LIN {X 0,Y 465.142,Z 330.415,A -85,B 0,C 180,E1 -14982.121,E2 -14982.121} C_VEL
LIN {X 0,Y 468.433,Z 327.76,A -85,B 0,C 180,E1 -14982.417,E2 -14982.417} C_VEL
LIN {X 0,Y 473.439,Z 325.91,A -85,B 0,C 180,E1 -14983.014,E2 -14983.014} C_VEL
LIN {X 0,Y 476.656,Z 325.887,A -85,B 0,C 180,E1 -14983.476,E2 -14983.476} C_VEL
LIN {X 0,Y 482.321,Z 341.882,A -85,B 0,C 180,E1 -14985.491,E2 -14985.491} C_VEL
LIN {X 0,Y 481.738,Z 369.053,A -85,B 0,C 180,E1 -14987.374,E2 -14987.374} C_VEL
LIN {X 0,Y 476.688,Z 392.56,A -85,B 0,C 180,E1 -14988.235,E2 -14988.235} C_VEL
LIN {X 0,Y 472.973,Z 475.5,A -85,B 0,C 180,E1 -14989.59,E2 -14989.59} C_VEL
LIN {X 0,Y 468.98,Z 538.697,A -85,B 0,C 180,E1 -14990.825,E2 -14990.825} C_VEL
LIN {X 0,Y 463.668,Z 606.761,A -85,B 0,C 180,E1 -14992.375,E2 -14992.375} C_VEL
LIN {X 0,Y 460.239,Z 651.951,A -85,B 0,C 180,E1 -14993.579,E2 -14993.579} C_VEL
LIN {X 0,Y 458.656,Z 674.727,A -85,B 0,C 180,E1 -14994.346,E2 -14994.346} C_VEL
LIN {X 0,Y 456.595,Z 696.121,A -85,B 0,C 180,E1 -14995.294,E2 -14995.294} C_VEL
LIN {X 0,Y 454.077,Z 716.813,A -85,B 0,C 180,E1 -14996.447,E2 -14996.447} C_VEL
LIN {X 0,Y 452.526,Z 727.999,A -85,B 0,C 180,E1 -14997.18,E2 -14997.18} C_VEL
LIN {X 0,Y 450.699,Z 734.854,A -85,B 0,C 180,E1 -14997.592,E2 -14997.592} C_VEL
LIN {X 0,Y 442.928,Z 751.978,A -85,B 0,C 180,E1 -14998.507,E2 -14998.507} C_VEL
LIN {X 0,Y 440.936,Z 758.361,A -85,B 0,C 180,E1 -14999.008,E2 -14999.008} C_VEL
LIN {X 0,Y 437.431,Z 776.665,A -85,B 0,C 180,E1 -15000.864,E2 -15000.864} C_VEL
LIN {X 0,Y 433.922,Z 793.74,A -85,B 0,C 180,E1 -15002.928,E2 -15002.928} C_VEL
LIN {X 0,Y 430.589,Z 809.209,A -85,B 0,C 180,E1 -15005.146,E2 -15005.146} C_VEL
LIN {X 0,Y 427.587,Z 822.933,A -85,B 0,C 180,E1 -15007.472,E2 -15007.472} C_VEL
LIN {X 0,Y 424.814,Z 835.676,A -85,B 0,C 180,E1 -15010.045,E2 -15010.045} C_VEL
LIN {X 0,Y 422.444,Z 846.943,A -85,B 0,C 180,E1 -15012.79,E2 -15012.79} C_VEL
LIN {X 0,Y 420.551,Z 856.578,A -85,B 0,C 180,E1 -15015.684,E2 -15015.684} C_VEL
LIN {X 0,Y 419.196,Z 864.185,A -85,B 0,C 180,E1 -15018.581,E2 -15018.581} C_VEL
LIN {X 0,Y 418.339,Z 869.705,A -85,B 0,C 180,E1 -15021.339,E2 -15021.339} C_VEL
LIN {X 0,Y 417.806,Z 873.843,A -85,B 0,C 180,E1 -15024.231,E2 -15024.231} C_VEL
LIN {X 0,Y 417.544,Z 876.277,A -85,B 0,C 180,E1 -15026.98,E2 -15026.98} C_VEL
LIN {X 0,Y 417.459,Z 877.198,A -85,B 0,C 180,E1 -15029.863,E2 -15029.863} C_VEL
LIN {X 0,Y 417.51,Z 876.519,A -85,B 0,C 180,E1 -15032.608,E2 -15032.608} C_VEL
LIN {X 0,Y 417.764,Z 874.258,A -85,B 0,C 180,E1 -15035.494,E2 -15035.494} C_VEL
LIN {X 0,Y 418.227,Z 870.613,A -85,B 0,C 180,E1 -15038.247,E2 -15038.247} C_VEL
LIN {X 0,Y 419.071,Z 865.05,A -85,B 0,C 180,E1 -15041.143,E2 -15041.143} C_VEL
LIN {X 0,Y 420.276,Z 858.016,A -85,B 0,C 180,E1 -15043.906,E2 -15043.906} C_VEL
LIN {X 0,Y 421.971,Z 849.236,A -85,B 0,C 180,E1 -15046.661,E2 -15046.661} C_VEL
LIN {X 0,Y 424.212,Z 838.486,A -85,B 0,C 180,E1 -15049.411,E2 -15049.411} C_VEL
LIN {X 0,Y 426.882,Z 826.191,A -85,B 0,C 180,E1 -15052.01,E2 -15052.01} C_VEL
LIN {X 0,Y 429.757,Z 813.215,A -85,B 0,C 180,E1 -15054.319,E2 -15054.319} C_VEL
LIN {X 0,Y 433.075,Z 797.976,A -85,B 0,C 180,E1 -15056.61,E2 -15056.61} C_VEL
LIN {X 0,Y 436.501,Z 781.676,A -85,B 0,C 180,E1 -15058.677,E2 -15058.677} C_VEL
LIN {X 0,Y 440.028,Z 763.676,A -85,B 0,C 180,E1 -15060.597,E2 -15060.597} C_VEL
LIN {X 0,Y 443.454,Z 744.549,A -85,B 0,C 180,E1 -15062.302,E2 -15062.302} C_VEL
LIN {X 0,Y 446.63,Z 724.241,A -85,B 0,C 180,E1 -15063.802,E2 -15063.802} C_VEL
LIN {X 0,Y 449.363,Z 703.738,A -85,B 0,C 180,E1 -15065.035,E2 -15065.035} C_VEL
LIN {X 0,Y 451.591,Z 682.841,A -85,B 0,C 180,E1 -15066.044,E2 -15066.044} C_VEL
LIN {X 0,Y 453.312,Z 661.563,A -85,B 0,C 180,E1 -15066.837,E2 -15066.837} C_VEL
LIN {X 0,Y 456.433,Z 619.357,A -85,B 0,C 180,E1 -15068.038,E2 -15068.038} C_VEL
LIN {X 0,Y 462.05,Z 551.52,A -85,B 0,C 180,E1 -15069.647,E2 -15069.647} C_VEL
LIN {X 0,Y 466.509,Z 485.901,A -85,B 0,C 180,E1 -15070.975,E2 -15070.975} C_VEL
LIN {X 0,Y 469.976,Z 414.611,A -85,B 0,C 180,E1 -15072.175,E2 -15072.175} C_VEL
LIN {X 0,Y 471.052,Z 393.311,A -85,B 0,C 180,E1 -15072.537,E2 -15072.537} C_VEL
LIN {X 0,Y 476.185,Z 369.743,A -85,B 0,C 180,E1 -15073.439,E2 -15073.439} C_VEL
LIN {X 0,Y 476.556,Z 345.293,A -85,B 0,C 180,E1 -15075.172,E2 -15075.172} C_VEL
LIN {X 0,Y 469.126,Z 324.998,A -85,B 0,C 180,E1 -15077.825,E2 -15077.825} C_VEL
LIN {X 0,Y 462.685,Z 309.482,A -85,B 0,C 180,E1 -15080.071,E2 -15080.071} C_VEL
LIN {X 0,Y 456.022,Z 295.191,A -85,B 0,C 180,E1 -15082.33,E2 -15082.33} C_VEL
LIN {X 0,Y 447.821,Z 279.246,A -85,B 0,C 180,E1 -15085.138,E2 -15085.138} C_VEL
LIN {X 0,Y 439.708,Z 265.393,A -85,B 0,C 180,E1 -15087.851,E2 -15087.851} C_VEL
LIN {X 0,Y 435.741,Z 259.224,A -85,B 0,C 180,E1 -15089.222,E2 -15089.222} C_VEL
LIN {X 0,Y 433.247,Z 255.233,A -85,B 0,C 180,E1 -15090.099,E2 -15090.099} C_VEL
LIN {X 0,Y 430.503,Z 250.807,A -85,B 0,C 180,E1 -15091.112,E2 -15091.112} C_VEL
LIN {X 0,Y 427.306,Z 246.461,A -85,B 0,C 180,E1 -15092.247,E2 -15092.247} C_VEL
LIN {X 0,Y 426.374,Z 244.715,A -85,B 0,C 180,E1 -15092.636,E2 -15092.636} C_VEL
LIN {X 0,Y 423.833,Z 241.89,A -85,B 0,C 180,E1 -15093.52,E2 -15093.52} C_VEL
LIN {X 0,Y 422.541,Z 239.071,A -85,B 0,C 180,E1 -15094.113,E2 -15094.113} C_VEL
LIN {X 0,Y 419.683,Z 236.312,A -85,B 0,C 180,E1 -15095.133,E2 -15095.133} C_VEL
LIN {X 0,Y 418.562,Z 233.254,A -85,B 0,C 180,E1 -15095.739,E2 -15095.739} C_VEL
LIN {X 0,Y 418.538,Z 233.089,A -85,B 0,C 180,E1 -15099.47,E2 -15099.47} C_VEL
LIN {X 0,Y 418.533,Z 233.058,A -85,B 0,C 180,E1 -15103.34,E2 -15103.34} C_VEL
LIN {X 0,Y 418.534,Z 233.043,A -85,B 0,C 180,E1 -15107.163,E2 -15107.163} C_VEL
LIN {X 0,Y 418.54,Z 233.095,A -85,B 0,C 180,E1 -15111.067,E2 -15111.067} C_VEL
LIN {X 0,Y 418.532,Z 233.045,A -85,B 0,C 180,E1 -15114.929,E2 -15114.929} C_VEL
LIN {X 0,Y 418.529,Z 233.064,A -85,B 0,C 180,E1 -15118.768,E2 -15118.768} C_VEL
LIN {X 0,Y 418.52,Z 233.07,A -85,B 0,C 180,E1 -15122.602,E2 -15122.602} C_VEL
LIN {X 0,Y 418.513,Z 233.043,A -85,B 0,C 180,E1 -15126.447,E2 -15126.447} C_VEL
LIN {X 0,Y 418.52,Z 233.1,A -85,B 0,C 180,E1 -15130.322,E2 -15130.322} C_VEL
LIN {X 0,Y 418.52,Z 233.096,A -85,B 0,C 180,E1 -15134.246,E2 -15134.246} C_VEL
LIN {X 0,Y 418.525,Z 233.086,A -85,B 0,C 180,E1 -15138.094,E2 -15138.094} C_VEL
LIN {X 0,Y 418.533,Z 233.168,A -85,B 0,C 180,E1 -15138.928,E2 -15138.928} C_VEL
LIN {X 0,Y 419.796,Z 236.493,A -85,B 0,C 180,E1 -15139.624,E2 -15139.624} C_VEL
LIN {X 0,Y 421.099,Z 238.531,A -85,B 0,C 180,E1 -15140.139,E2 -15140.139} C_VEL
LIN {X 0,Y 423.255,Z 242.427,A -85,B 0,C 180,E1 -15141.044,E2 -15141.044} C_VEL
LIN {X 0,Y 430.88,Z 257.106,A -85,B 0,C 180,E1 -15144.252,E2 -15144.252} C_VEL
LIN {X 0,Y 439.608,Z 273.969,A -85,B 0,C 180,E1 -15147.646,E2 -15147.646} C_VEL
LIN {X 0,Y 449.782,Z 294.439,A -85,B 0,C 180,E1 -15151.345,E2 -15151.345} C_VEL
LIN {X 0,Y 459.809,Z 315.283,A -85,B 0,C 180,E1 -15154.732,E2 -15154.732} C_VEL
LIN {X 0,Y 464.788,Z 325.491,A -85,B 0,C 180,E1 -15156.233,E2 -15156.233} C_VEL
LIN {X 0,Y 480.323,Z 350.017,A -85,B 0,C 180,E1 -15158.475,E2 -15158.475} C_VEL
LIN {X 0,Y 480.604,Z 356.269,A -85,B 0,C 180,E1 -15158.658,E2 -15158.658} C_VEL
LIN {X 0,Y 466.182,Z 601.705,A -85,B 0,C 180,E1 -15163.233,E2 -15163.233} C_VEL
LIN {X 0,Y 461.361,Z 693.458,A -85,B 0,C 180,E1 -15164.963,E2 -15164.963} C_VEL
LIN {X 0,Y 459.117,Z 717.943,A -85,B 0,C 180,E1 -15165.63,E2 -15165.63} C_VEL
LIN {X 0,Y 456.209,Z 743.457,A -85,B 0,C 180,E1 -15166.552,E2 -15166.552} C_VEL
LIN {X 0,Y 453.173,Z 765.825,A -85,B 0,C 180,E1 -15167.576,E2 -15167.576} C_VEL
LIN {X 0,Y 449.498,Z 789.387,A -85,B 0,C 180,E1 -15168.904,E2 -15168.904} C_VEL
LIN {X 0,Y 445.801,Z 811.052,A -85,B 0,C 180,E1 -15170.358,E2 -15170.358} C_VEL
LIN {X 0,Y 441.915,Z 831.707,A -85,B 0,C 180,E1 -15172.017,E2 -15172.017} C_VEL
LIN {X 0,Y 437.866,Z 852.231,A -85,B 0,C 180,E1 -15173.938,E2 -15173.938} C_VEL
LIN {X 0,Y 434.211,Z 870.106,A -85,B 0,C 180,E1 -15175.894,E2 -15175.894} C_VEL
LIN {X 0,Y 430.262,Z 889.208,A -85,B 0,C 180,E1 -15178.318,E2 -15178.318} C_VEL
LIN {X 0,Y 426.966,Z 905.358,A -85,B 0,C 180,E1 -15180.696,E2 -15180.696} C_VEL
LIN {X 0,Y 423.914,Z 920.881,A -85,B 0,C 180,E1 -15183.375,E2 -15183.375} C_VEL
LIN {X 0,Y 421.465,Z 934.402,A -85,B 0,C 180,E1 -15186.066,E2 -15186.066} C_VEL
LIN {X 0,Y 419.512,Z 946.432,A -85,B 0,C 180,E1 -15188.906,E2 -15188.906} C_VEL
LIN {X 0,Y 418.139,Z 956.77,A -85,B 0,C 180,E1 -15191.744,E2 -15191.744} C_VEL
LIN {X 0,Y 417.219,Z 965.635,A -85,B 0,C 180,E1 -15194.715,E2 -15194.715} C_VEL
LIN {X 0,Y 416.734,Z 972.905,A -85,B 0,C 180,E1 -15197.67,E2 -15197.67} C_VEL
LIN {X 0,Y 416.585,Z 978.694,A -85,B 0,C 180,E1 -15200.746,E2 -15200.746} C_VEL
LIN {X 0,Y 416.629,Z 982.359,A -85,B 0,C 180,E1 -15203.385,E2 -15203.385} C_VEL
LIN {X 0,Y 416.736,Z 985.143,A -85,B 0,C 180,E1 -15206.423,E2 -15206.423} C_VEL
LIN {X 0,Y 416.795,Z 986.147,A -85,B 0,C 180,E1 -15209.313,E2 -15209.313} C_VEL
LIN {X 0,Y 416.792,Z 985.858,A -85,B 0,C 180,E1 -15211.925,E2 -15211.925} C_VEL
LIN {X 0,Y 416.657,Z 984.108,A -85,B 0,C 180,E1 -15214.956,E2 -15214.956} C_VEL
LIN {X 0,Y 416.576,Z 980.619,A -85,B 0,C 180,E1 -15218.003,E2 -15218.003} C_VEL
LIN {X 0,Y 416.588,Z 976.376,A -85,B 0,C 180,E1 -15220.65,E2 -15220.65} C_VEL
LIN {X 0,Y 416.89,Z 969.637,A -85,B 0,C 180,E1 -15223.878,E2 -15223.878} C_VEL
LIN {X 0,Y 417.582,Z 961.789,A -85,B 0,C 180,E1 -15226.842,E2 -15226.842} C_VEL
LIN {X 0,Y 418.851,Z 951.921,A -85,B 0,C 180,E1 -15229.961,E2 -15229.961} C_VEL
LIN {X 0,Y 420.695,Z 940.588,A -85,B 0,C 180,E1 -15232.941,E2 -15232.941} C_VEL
LIN {X 0,Y 423.28,Z 927.489,A -85,B 0,C 180,E1 -15235.914,E2 -15235.914} C_VEL
LIN {X 0,Y 426.486,Z 912.889,A -85,B 0,C 180,E1 -15238.736,E2 -15238.736} C_VEL
LIN {X 0,Y 430.666,Z 895.41,A -85,B 0,C 180,E1 -15241.649,E2 -15241.649} C_VEL
LIN {X 0,Y 435.032,Z 878.269,A -85,B 0,C 180,E1 -15244.112,E2 -15244.112} C_VEL
LIN {X 0,Y 439.906,Z 859.257,A -85,B 0,C 180,E1 -15246.461,E2 -15246.461} C_VEL
LIN {X 0,Y 445.064,Z 839.529,A -85,B 0,C 180,E1 -15248.572,E2 -15248.572} C_VEL
LIN {X 0,Y 450.442,Z 818.443,A -85,B 0,C 180,E1 -15250.488,E2 -15250.488} C_VEL
LIN {X 0,Y 455.993,Z 795.957,A -85,B 0,C 180,E1 -15252.228,E2 -15252.228} C_VEL
LIN {X 0,Y 461.455,Z 772.834,A -85,B 0,C 180,E1 -15253.727,E2 -15253.727} C_VEL
LIN {X 0,Y 466.711,Z 748.74,A -85,B 0,C 180,E1 -15255.009,E2 -15255.009} C_VEL
LIN {X 0,Y 471.508,Z 724.263,A -85,B 0,C 180,E1 -15256.051,E2 -15256.051} C_VEL
LIN {X 0,Y 476.08,Z 697.875,A -85,B 0,C 180,E1 -15256.912,E2 -15256.912} C_VEL
LIN {X 0,Y 481.22,Z 660.217,A -85,B 0,C 180,E1 -15257.828,E2 -15257.828} C_VEL
LIN {X 0,Y 489.533,Z 604.335,A -85,B 0,C 180,E1 -15259.157,E2 -15259.157} C_VEL
LIN {X 0,Y 500.202,Z 547.443,A -85,B 0,C 180,E1 -15260.549,E2 -15260.549} C_VEL
LIN {X 0,Y 508.93,Z 508.11,A -85,B 0,C 180,E1 -15261.532,E2 -15261.532} C_VEL
LIN {X 0,Y 504.603,Z 526.167,A -85,B 0,C 180,E1 -15262.441,E2 -15262.441} C_VEL
LIN {X 0,Y 481.706,Z 630.182,A -85,B 0,C 180,E1 -15265.508,E2 -15265.508} C_VEL
LIN {X 0,Y 469.101,Z 693.847,A -85,B 0,C 180,E1 -15267.556,E2 -15267.556} C_VEL
LIN {X 0,Y 463.766,Z 717.456,A -85,B 0,C 180,E1 -15268.55,E2 -15268.55} C_VEL
LIN {X 0,Y 458.09,Z 740.922,A -85,B 0,C 180,E1 -15269.815,E2 -15269.815} C_VEL
LIN {X 0,Y 452.388,Z 763.754,A -85,B 0,C 180,E1 -15271.339,E2 -15271.339} C_VEL
LIN {X 0,Y 447.011,Z 785.108,A -85,B 0,C 180,E1 -15273.066,E2 -15273.066} C_VEL
LIN {X 0,Y 442.238,Z 804.171,A -85,B 0,C 180,E1 -15274.917,E2 -15274.917} C_VEL
LIN {X 0,Y 437.83,Z 821.686,A -85,B 0,C 180,E1 -15276.942,E2 -15276.942} C_VEL
LIN {X 0,Y 433.913,Z 837.047,A -85,B 0,C 180,E1 -15279.073,E2 -15279.073} C_VEL
LIN {X 0,Y 430.445,Z 850.31,A -85,B 0,C 180,E1 -15281.303,E2 -15281.303} C_VEL
LIN {X 0,Y 427.606,Z 860.933,A -85,B 0,C 180,E1 -15283.481,E2 -15283.481} C_VEL
LIN {X 0,Y 425.193,Z 869.743,A -85,B 0,C 180,E1 -15285.705,E2 -15285.705} C_VEL
LIN {X 0,Y 423.039,Z 877.204,A -85,B 0,C 180,E1 -15288.133,E2 -15288.133} C_VEL
LIN {X 0,Y 421.42,Z 882.367,A -85,B 0,C 180,E1 -15290.44,E2 -15290.44} C_VEL
LIN {X 0,Y 420.191,Z 885.911,A -85,B 0,C 180,E1 -15292.755,E2 -15292.755} C_VEL
LIN {X 0,Y 419.213,Z 887.887,A -85,B 0,C 180,E1 -15295.211,E2 -15295.211} C_VEL
LIN {X 0,Y 418.581,Z 888.17,A -85,B 0,C 180,E1 -15297.536,E2 -15297.536} C_VEL
LIN {X 0,Y 418.161,Z 886.727,A -85,B 0,C 180,E1 -15300,E2 -15300} C_VEL
LIN {X 0,Y 417.948,Z 883.54,A -85,B 0,C 180,E1 -15302.468,E2 -15302.468} C_VEL
LIN {X 0,Y 417.955,Z 878.555,A -85,B 0,C 180,E1 -15304.941,E2 -15304.941} C_VEL
LIN {X 0,Y 418.197,Z 871.701,A -85,B 0,C 180,E1 -15307.418,E2 -15307.418} C_VEL
LIN {X 0,Y 418.711,Z 862.825,A -85,B 0,C 180,E1 -15309.901,E2 -15309.901} C_VEL
LIN {X 0,Y 419.516,Z 852.331,A -85,B 0,C 180,E1 -15312.255,E2 -15312.255} C_VEL
LIN {X 0,Y 420.579,Z 840.438,A -85,B 0,C 180,E1 -15314.456,E2 -15314.456} C_VEL
LIN {X 0,Y 421.988,Z 826.127,A -85,B 0,C 180,E1 -15316.661,E2 -15316.661} C_VEL
LIN {X 0,Y 423.658,Z 810.108,A -85,B 0,C 180,E1 -15318.722,E2 -15318.722} C_VEL
LIN {X 0,Y 425.556,Z 792.28,A -85,B 0,C 180,E1 -15320.637,E2 -15320.637} C_VEL
LIN {X 0,Y 427.535,Z 773.248,A -85,B 0,C 180,E1 -15322.337,E2 -15322.337} C_VEL
LIN {X 0,Y 429.463,Z 754.068,A -85,B 0,C 180,E1 -15323.753,E2 -15323.753} C_VEL
LIN {X 0,Y 431.425,Z 733.007,A -85,B 0,C 180,E1 -15325.014,E2 -15325.014} C_VEL
LIN {X 0,Y 433.222,Z 711.178,A -85,B 0,C 180,E1 -15326.047,E2 -15326.047} C_VEL
LIN {X 0,Y 434.895,Z 687.679,A -85,B 0,C 180,E1 -15326.879,E2 -15326.879} C_VEL
LIN {X 0,Y 437.042,Z 646.566,A -85,B 0,C 180,E1 -15327.878,E2 -15327.878} C_VEL
LIN {X 0,Y 444.712,Z 506.022,A -85,B 0,C 180,E1 -15331.093,E2 -15331.093} C_VEL
LIN {X 0,Y 439.779,Z 438.733,A -85,B 0,C 180,E1 -15333.306,E2 -15333.306} C_VEL
LIN {X 0,Y 445.969,Z 387.644,A -85,B 0,C 180,E1 -15337.489,E2 -15337.489} C_VEL
LIN {X 0,Y 451.691,Z 344.172,A -85,B 0,C 180,E1 -15341.064,E2 -15341.064} C_VEL
LIN {X 0,Y 453.675,Z 344.144,A -85,B 0,C 180,E1 -15341.391,E2 -15341.391} C_VEL
LIN {X 0,Y 456.593,Z 342.501,A -85,B 0,C 180,E1 -15341.738,E2 -15341.738} C_VEL
LIN {X 0,Y 459.898,Z 339.563,A -85,B 0,C 180,E1 -15342.04,E2 -15342.04} C_VEL
LIN {X 0,Y 463.43,Z 338.215,A -85,B 0,C 180,E1 -15342.48,E2 -15342.48} C_VEL
LIN {X 0,Y 468.257,Z 334.771,A -85,B 0,C 180,E1 -15342.936,E2 -15342.936} C_VEL
LIN {X 0,Y 472.208,Z 333.263,A -85,B 0,C 180,E1 -15343.4,E2 -15343.4} C_VEL
LIN {X 0,Y 476.586,Z 346.018,A -85,B 0,C 180,E1 -15345.006,E2 -15345.006} C_VEL
LIN {X 0,Y 476.081,Z 370.363,A -85,B 0,C 180,E1 -15346.707,E2 -15346.707} C_VEL
LIN {X 0,Y 470.702,Z 395.368,A -85,B 0,C 180,E1 -15347.619,E2 -15347.619} C_VEL
LIN {X 0,Y 466.885,Z 477.849,A -85,B 0,C 180,E1 -15348.979,E2 -15348.979} C_VEL
LIN {X 0,Y 462.789,Z 540.682,A -85,B 0,C 180,E1 -15350.221,E2 -15350.221} C_VEL
LIN {X 0,Y 457.359,Z 607.896,A -85,B 0,C 180,E1 -15351.773,E2 -15351.773} C_VEL
LIN {X 0,Y 453.808,Z 652.838,A -85,B 0,C 180,E1 -15352.992,E2 -15352.992} C_VEL
LIN {X 0,Y 452.145,Z 676.013,A -85,B 0,C 180,E1 -15353.781,E2 -15353.781} C_VEL
LIN {X 0,Y 450.073,Z 696.948,A -85,B 0,C 180,E1 -15354.716,E2 -15354.716} C_VEL
LIN {X 0,Y 447.372,Z 718.396,A -85,B 0,C 180,E1 -15355.927,E2 -15355.927} C_VEL
LIN {X 0,Y 444.251,Z 739.171,A -85,B 0,C 180,E1 -15357.381,E2 -15357.381} C_VEL
LIN {X 0,Y 440.936,Z 758.361,A -85,B 0,C 180,E1 -15359.008,E2 -15359.008} C_VEL
LIN {X 0,Y 438.931,Z 764.725,A -85,B 0,C 180,E1 -15359.533,E2 -15359.533} C_VEL
LIN {X 0,Y 430.735,Z 780.584,A -85,B 0,C 180,E1 -15360.754,E2 -15360.754} C_VEL
LIN {X 0,Y 428.649,Z 786.403,A -85,B 0,C 180,E1 -15361.374,E2 -15361.374} C_VEL
LIN {X 0,Y 425.203,Z 802.108,A -85,B 0,C 180,E1 -15363.462,E2 -15363.462} C_VEL
LIN {X 0,Y 421.843,Z 816.908,A -85,B 0,C 180,E1 -15365.791,E2 -15365.791} C_VEL
LIN {X 0,Y 418.786,Z 830.224,A -85,B 0,C 180,E1 -15368.28,E2 -15368.28} C_VEL
LIN {X 0,Y 415.99,Z 842.599,A -85,B 0,C 180,E1 -15371.065,E2 -15371.065} C_VEL
LIN {X 0,Y 413.787,Z 852.799,A -85,B 0,C 180,E1 -15373.866,E2 -15373.866} C_VEL
LIN {X 0,Y 412.078,Z 861.435,A -85,B 0,C 180,E1 -15376.815,E2 -15376.815} C_VEL
LIN {X 0,Y 410.917,Z 867.862,A -85,B 0,C 180,E1 -15379.626,E2 -15379.626} C_VEL
LIN {X 0,Y 410.156,Z 872.891,A -85,B 0,C 180,E1 -15382.576,E2 -15382.576} C_VEL
LIN {X 0,Y 409.729,Z 876.243,A -85,B 0,C 180,E1 -15385.521,E2 -15385.521} C_VEL
LIN {X 0,Y 409.54,Z 877.981,A -85,B 0,C 180,E1 -15388.461,E2 -15388.461} C_VEL
LIN {X 0,Y 409.523,Z 878.039,A -85,B 0,C 180,E1 -15391.259,E2 -15391.259} C_VEL
LIN {X 0,Y 409.692,Z 876.537,A -85,B 0,C 180,E1 -15394.199,E2 -15394.199} C_VEL
LIN {X 0,Y 410.094,Z 873.424,A -85,B 0,C 180,E1 -15397.143,E2 -15397.143} C_VEL
LIN {X 0,Y 410.768,Z 868.937,A -85,B 0,C 180,E1 -15399.952,E2 -15399.952} C_VEL
LIN {X 0,Y 411.91,Z 862.424,A -85,B 0,C 180,E1 -15402.904,E2 -15402.904} C_VEL
LIN {X 0,Y 413.462,Z 854.365,A -85,B 0,C 180,E1 -15405.74,E2 -15405.74} C_VEL
LIN {X 0,Y 415.547,Z 844.595,A -85,B 0,C 180,E1 -15408.519,E2 -15408.519} C_VEL
LIN {X 0,Y 418.086,Z 833.296,A -85,B 0,C 180,E1 -15411.17,E2 -15411.17} C_VEL
LIN {X 0,Y 421.02,Z 820.573,A -85,B 0,C 180,E1 -15413.663,E2 -15413.663} C_VEL
LIN {X 0,Y 424.266,Z 806.441,A -85,B 0,C 180,E1 -15415.999,E2 -15415.999} C_VEL
LIN {X 0,Y 427.748,Z 790.854,A -85,B 0,C 180,E1 -15418.176,E2 -15418.176} C_VEL
LIN {X 0,Y 431.38,Z 773.694,A -85,B 0,C 180,E1 -15420.197,E2 -15420.197} C_VEL
LIN {X 0,Y 434.929,Z 755.568,A -85,B 0,C 180,E1 -15421.992,E2 -15421.992} C_VEL
LIN {X 0,Y 438.301,Z 736.243,A -85,B 0,C 180,E1 -15423.588,E2 -15423.588} C_VEL
LIN {X 0,Y 441.375,Z 715.92,A -85,B 0,C 180,E1 -15424.97,E2 -15424.97} C_VEL
LIN {X 0,Y 443.968,Z 695.234,A -85,B 0,C 180,E1 -15426.109,E2 -15426.109} C_VEL
LIN {X 0,Y 446.008,Z 674.403,A -85,B 0,C 180,E1 -15427.017,E2 -15427.017} C_VEL
LIN {X 0,Y 447.966,Z 647.329,A -85,B 0,C 180,E1 -15427.907,E2 -15427.907} C_VEL
LIN {X 0,Y 452.25,Z 596.981,A -85,B 0,C 180,E1 -15429.247,E2 -15429.247} C_VEL
LIN {X 0,Y 457.529,Z 532.097,A -85,B 0,C 180,E1 -15430.727,E2 -15430.727} C_VEL
LIN {X 0,Y 461.644,Z 467.647,A -85,B 0,C 180,E1 -15431.974,E2 -15431.974} C_VEL
LIN {X 0,Y 465.122,Z 396.05,A -85,B 0,C 180,E1 -15433.169,E2 -15433.169} C_VEL
LIN {X 0,Y 470.511,Z 371.711,A -85,B 0,C 180,E1 -15434.086,E2 -15434.086} C_VEL
LIN {X 0,Y 470.855,Z 349.322,A -85,B 0,C 180,E1 -15435.681,E2 -15435.681} C_VEL
LIN {X 0,Y 463.855,Z 330.038,A -85,B 0,C 180,E1 -15438.234,E2 -15438.234} C_VEL
LIN {X 0,Y 456.491,Z 312.145,A -85,B 0,C 180,E1 -15440.888,E2 -15440.888} C_VEL
LIN {X 0,Y 448.714,Z 295.881,A -85,B 0,C 180,E1 -15443.555,E2 -15443.555} C_VEL
LIN {X 0,Y 441.192,Z 281.498,A -85,B 0,C 180,E1 -15446.194,E2 -15446.194} C_VEL
LIN {X 0,Y 434.542,Z 270.327,A -85,B 0,C 180,E1 -15448.511,E2 -15448.511} C_VEL
LIN {X 0,Y 429.661,Z 262.251,A -85,B 0,C 180,E1 -15450.285,E2 -15450.285} C_VEL
LIN {X 0,Y 426.904,Z 258.059,A -85,B 0,C 180,E1 -15451.305,E2 -15451.305} C_VEL
LIN {X 0,Y 423.194,Z 252.399,A -85,B 0,C 180,E1 -15452.718,E2 -15452.718} C_VEL
LIN {X 0,Y 419.793,Z 247.902,A -85,B 0,C 180,E1 -15454.007,E2 -15454.007} C_VEL
LIN {X 0,Y 418.942,Z 246.069,A -85,B 0,C 180,E1 -15454.406,E2 -15454.406} C_VEL
LIN {X 0,Y 416.059,Z 242.908,A -85,B 0,C 180,E1 -15455.508,E2 -15455.508} C_VEL
LIN {X 0,Y 414.671,Z 240.056,A -85,B 0,C 180,E1 -15456.178,E2 -15456.178} C_VEL
LIN {X 0,Y 411.827,Z 237.422,A -85,B 0,C 180,E1 -15457.291,E2 -15457.291} C_VEL
LIN {X 0,Y 410.633,Z 234.295,A -85,B 0,C 180,E1 -15457.976,E2 -15457.976} C_VEL
LIN {X 0,Y 410.594,Z 234.03,A -85,B 0,C 180,E1 -15461.838,E2 -15461.838} C_VEL
LIN {X 0,Y 410.604,Z 234.058,A -85,B 0,C 180,E1 -15465.762,E2 -15465.762} C_VEL
LIN {X 0,Y 410.596,Z 234.057,A -85,B 0,C 180,E1 -15469.76,E2 -15469.76} C_VEL
LIN {X 0,Y 410.596,Z 234.027,A -85,B 0,C 180,E1 -15473.709,E2 -15473.709} C_VEL
LIN {X 0,Y 410.601,Z 234.083,A -85,B 0,C 180,E1 -15477.627,E2 -15477.627} C_VEL
LIN {X 0,Y 410.597,Z 234.031,A -85,B 0,C 180,E1 -15481.535,E2 -15481.535} C_VEL
LIN {X 0,Y 410.599,Z 234.046,A -85,B 0,C 180,E1 -15485.45,E2 -15485.45} C_VEL
LIN {X 0,Y 410.602,Z 234.061,A -85,B 0,C 180,E1 -15489.39,E2 -15489.39} C_VEL
LIN {X 0,Y 410.605,Z 234.083,A -85,B 0,C 180,E1 -15493.376,E2 -15493.376} C_VEL
LIN {X 0,Y 410.601,Z 234.084,A -85,B 0,C 180,E1 -15497.283,E2 -15497.283} C_VEL
LIN {X 0,Y 410.633,Z 234.282,A -85,B 0,C 180,E1 -15497.538,E2 -15497.538} C_VEL
LIN {X 0,Y 411.874,Z 237.541,A -85,B 0,C 180,E1 -15498.25,E2 -15498.25} C_VEL
LIN {X 0,Y 413.191,Z 239.4,A -85,B 0,C 180,E1 -15498.775,E2 -15498.775} C_VEL
LIN {X 0,Y 415.204,Z 243.299,A -85,B 0,C 180,E1 -15499.703,E2 -15499.703} C_VEL
LIN {X 0,Y 420.886,Z 254.249,A -85,B 0,C 180,E1 -15502.193,E2 -15502.193} C_VEL
LIN {X 0,Y 427.8,Z 267.468,A -85,B 0,C 180,E1 -15505.027,E2 -15505.027} C_VEL
LIN {X 0,Y 436.306,Z 284.141,A -85,B 0,C 180,E1 -15508.32,E2 -15508.32} C_VEL
LIN {X 0,Y 446.297,Z 304.362,A -85,B 0,C 180,E1 -15511.92,E2 -15511.92} C_VEL
LIN {X 0,Y 456.718,Z 326.072,A -85,B 0,C 180,E1 -15515.366,E2 -15515.366} C_VEL
LIN {X 0,Y 474.355,Z 353.885,A -85,B 0,C 180,E1 -15517.968,E2 -15517.968} C_VEL
LIN {X 0,Y 474.205,Z 360.312,A -85,B 0,C 180,E1 -15518.117,E2 -15518.117} C_VEL
LIN {X 0,Y 459.21,Z 606.522,A -85,B 0,C 180,E1 -15522.784,E2 -15522.784} C_VEL
LIN {X 0,Y 454.457,Z 693.43,A -85,B 0,C 180,E1 -15524.457,E2 -15524.457} C_VEL
LIN {X 0,Y 452.163,Z 717.773,A -85,B 0,C 180,E1 -15525.131,E2 -15525.131} C_VEL
LIN {X 0,Y 449.295,Z 742.351,A -85,B 0,C 180,E1 -15526.025,E2 -15526.025} C_VEL
LIN {X 0,Y 446.278,Z 764.081,A -85,B 0,C 180,E1 -15527.025,E2 -15527.025} C_VEL
LIN {X 0,Y 442.507,Z 787.894,A -85,B 0,C 180,E1 -15528.37,E2 -15528.37} C_VEL
LIN {X 0,Y 438.714,Z 809.559,A -85,B 0,C 180,E1 -15529.835,E2 -15529.835} C_VEL
LIN {X 0,Y 434.774,Z 830.163,A -85,B 0,C 180,E1 -15531.499,E2 -15531.499} C_VEL
LIN {X 0,Y 430.744,Z 850.203,A -85,B 0,C 180,E1 -15533.375,E2 -15533.375} C_VEL
LIN {X 0,Y 426.766,Z 869.103,A -85,B 0,C 180,E1 -15535.459,E2 -15535.459} C_VEL
LIN {X 0,Y 422.811,Z 887.794,A -85,B 0,C 180,E1 -15537.853,E2 -15537.853} C_VEL
LIN {X 0,Y 419.509,Z 903.423,A -85,B 0,C 180,E1 -15540.18,E2 -15540.18} C_VEL
LIN {X 0,Y 416.377,Z 918.925,A -85,B 0,C 180,E1 -15542.854,E2 -15542.854} C_VEL
LIN {X 0,Y 413.922,Z 931.913,A -85,B 0,C 180,E1 -15545.45,E2 -15545.45} C_VEL
LIN {X 0,Y 411.744,Z 944.833,A -85,B 0,C 180,E1 -15548.488,E2 -15548.488} C_VEL
LIN {X 0,Y 410.284,Z 955.269,A -85,B 0,C 180,E1 -15551.382,E2 -15551.382} C_VEL
LIN {X 0,Y 409.272,Z 964.688,A -85,B 0,C 180,E1 -15554.556,E2 -15554.556} C_VEL
LIN {X 0,Y 408.776,Z 971.983,A -85,B 0,C 180,E1 -15557.57,E2 -15557.57} C_VEL
LIN {X 0,Y 408.629,Z 977.786,A -85,B 0,C 180,E1 -15560.706,E2 -15560.706} C_VEL
LIN {X 0,Y 408.681,Z 981.444,A -85,B 0,C 180,E1 -15563.397,E2 -15563.397} C_VEL
LIN {X 0,Y 408.797,Z 984.212,A -85,B 0,C 180,E1 -15566.494,E2 -15566.494} C_VEL
LIN {X 0,Y 408.855,Z 985.183,A -85,B 0,C 180,E1 -15569.44,E2 -15569.44} C_VEL
LIN {X 0,Y 408.837,Z 984.862,A -85,B 0,C 180,E1 -15572.102,E2 -15572.102} C_VEL
LIN {X 0,Y 408.69,Z 983.057,A -85,B 0,C 180,E1 -15575.194,E2 -15575.194} C_VEL
LIN {X 0,Y 408.594,Z 979.51,A -85,B 0,C 180,E1 -15578.302,E2 -15578.302} C_VEL
LIN {X 0,Y 408.613,Z 975.041,A -85,B 0,C 180,E1 -15581.108,E2 -15581.108} C_VEL
LIN {X 0,Y 408.992,Z 968.066,A -85,B 0,C 180,E1 -15584.44,E2 -15584.44} C_VEL
LIN {X 0,Y 409.782,Z 960.115,A -85,B 0,C 180,E1 -15587.465,E2 -15587.465} C_VEL
LIN {X 0,Y 411.287,Z 949.569,A -85,B 0,C 180,E1 -15590.79,E2 -15590.79} C_VEL
LIN {X 0,Y 413.253,Z 938.67,A -85,B 0,C 180,E1 -15593.681,E2 -15593.681} C_VEL
LIN {X 0,Y 416.402,Z 923.909,A -85,B 0,C 180,E1 -15597.017,E2 -15597.017} C_VEL
LIN {X 0,Y 419.914,Z 909.28,A -85,B 0,C 180,E1 -15599.846,E2 -15599.846} C_VEL
LIN {X 0,Y 424.304,Z 892.298,A -85,B 0,C 180,E1 -15602.66,E2 -15602.66} C_VEL
LIN {X 0,Y 429.296,Z 873.956,A -85,B 0,C 180,E1 -15605.284,E2 -15605.284} C_VEL
LIN {X 0,Y 434.639,Z 854.657,A -85,B 0,C 180,E1 -15607.646,E2 -15607.646} C_VEL
LIN {X 0,Y 440.371,Z 833.928,A -85,B 0,C 180,E1 -15609.814,E2 -15609.814} C_VEL
LIN {X 0,Y 445.99,Z 813.441,A -85,B 0,C 180,E1 -15611.663,E2 -15611.663} C_VEL
LIN {X 0,Y 451.965,Z 790.62,A -85,B 0,C 180,E1 -15613.387,E2 -15613.387} C_VEL
LIN {X 0,Y 457.815,Z 767.151,A -85,B 0,C 180,E1 -15614.866,E2 -15614.866} C_VEL
LIN {X 0,Y 463.428,Z 743.115,A -85,B 0,C 180,E1 -15616.107,E2 -15616.107} C_VEL
LIN {X 0,Y 468.675,Z 718.317,A -85,B 0,C 180,E1 -15617.125,E2 -15617.125} C_VEL
LIN {X 0,Y 473.177,Z 693.617,A -85,B 0,C 180,E1 -15617.9,E2 -15617.9} C_VEL
LIN {X 0,Y 485.132,Z 617.626,A -85,B 0,C 180,E1 -15619.751,E2 -15619.751} C_VEL
LIN {X 0,Y 496.148,Z 562.189,A -85,B 0,C 180,E1 -15621.116,E2 -15621.116} C_VEL
LIN {X 0,Y 502.171,Z 535.812,A -85,B 0,C 180,E1 -15621.777,E2 -15621.777} C_VEL
LIN {X 0,Y 478.06,Z 639.781,A -85,B 0,C 180,E1 -15624.851,E2 -15624.851} C_VEL
LIN {X 0,Y 466.558,Z 693.913,A -85,B 0,C 180,E1 -15626.607,E2 -15626.607} C_VEL
LIN {X 0,Y 460.795,Z 717.287,A -85,B 0,C 180,E1 -15627.59,E2 -15627.59} C_VEL
LIN {X 0,Y 454.74,Z 739.998,A -85,B 0,C 180,E1 -15628.814,E2 -15628.814} C_VEL
LIN {X 0,Y 448.459,Z 762.678,A -85,B 0,C 180,E1 -15630.332,E2 -15630.332} C_VEL
LIN {X 0,Y 442.189,Z 785.109,A -85,B 0,C 180,E1 -15632.164,E2 -15632.164} C_VEL
LIN {X 0,Y 436.82,Z 804.476,A -85,B 0,C 180,E1 -15634.074,E2 -15634.074} C_VEL
LIN {X 0,Y 432.024,Z 821.806,A -85,B 0,C 180,E1 -15636.107,E2 -15636.107} C_VEL
LIN {X 0,Y 427.866,Z 836.688,A -85,B 0,C 180,E1 -15638.187,E2 -15638.187} C_VEL
LIN {X 0,Y 424.085,Z 850.143,A -85,B 0,C 180,E1 -15640.439,E2 -15640.439} C_VEL
LIN {X 0,Y 420.685,Z 861.897,A -85,B 0,C 180,E1 -15642.859,E2 -15642.859} C_VEL
LIN {X 0,Y 417.846,Z 871.334,A -85,B 0,C 180,E1 -15645.306,E2 -15645.306} C_VEL
LIN {X 0,Y 415.638,Z 878.281,A -85,B 0,C 180,E1 -15647.637,E2 -15647.637} C_VEL
LIN {X 0,Y 413.877,Z 883.502,A -85,B 0,C 180,E1 -15649.983,E2 -15649.983} C_VEL
LIN {X 0,Y 412.447,Z 887.202,A -85,B 0,C 180,E1 -15652.478,E2 -15652.478} C_VEL
LIN {X 0,Y 411.394,Z 889.136,A -85,B 0,C 180,E1 -15654.98,E2 -15654.98} C_VEL
LIN {X 0,Y 410.666,Z 889.291,A -85,B 0,C 180,E1 -15657.488,E2 -15657.488} C_VEL
LIN {X 0,Y 410.24,Z 887.847,A -85,B 0,C 180,E1 -15659.86,E2 -15659.86} C_VEL
LIN {X 0,Y 410.002,Z 884.604,A -85,B 0,C 180,E1 -15662.376,E2 -15662.376} C_VEL
LIN {X 0,Y 409.997,Z 879.569,A -85,B 0,C 180,E1 -15664.897,E2 -15664.897} C_VEL
LIN {X 0,Y 410.237,Z 872.646,A -85,B 0,C 180,E1 -15667.422,E2 -15667.422} C_VEL
LIN {X 0,Y 410.759,Z 863.693,A -85,B 0,C 180,E1 -15669.953,E2 -15669.953} C_VEL
LIN {X 0,Y 411.582,Z 853.184,A -85,B 0,C 180,E1 -15672.344,E2 -15672.344} C_VEL
LIN {X 0,Y 412.682,Z 841.23,A -85,B 0,C 180,E1 -15674.595,E2 -15674.595} C_VEL
LIN {X 0,Y 414.082,Z 827.361,A -85,B 0,C 180,E1 -15676.772,E2 -15676.772} C_VEL
LIN {X 0,Y 415.785,Z 811.363,A -85,B 0,C 180,E1 -15678.872,E2 -15678.872} C_VEL
LIN {X 0,Y 417.725,Z 793.581,A -85,B 0,C 180,E1 -15680.822,E2 -15680.822} C_VEL
LIN {X 0,Y 419.747,Z 774.635,A -85,B 0,C 180,E1 -15682.552,E2 -15682.552} C_VEL
LIN {X 0,Y 421.818,Z 754.622,A -85,B 0,C 180,E1 -15684.061,E2 -15684.061} C_VEL
LIN {X 0,Y 423.846,Z 733.462,A -85,B 0,C 180,E1 -15685.352,E2 -15685.352} C_VEL
LIN {X 0,Y 425.613,Z 712.677,A -85,B 0,C 180,E1 -15686.361,E2 -15686.361} C_VEL
LIN {X 0,Y 427.276,Z 690.14,A -85,B 0,C 180,E1 -15687.192,E2 -15687.192} C_VEL
LIN {X 0,Y 429.095,Z 657.974,A -85,B 0,C 180,E1 -15688.024,E2 -15688.024} C_VEL
LIN {X 0,Y 437.616,Z 506.725,A -85,B 0,C 180,E1 -15691.574,E2 -15691.574} C_VEL
LIN {X 0,Y 432.779,Z 437.458,A -85,B 0,C 180,E1 -15693.915,E2 -15693.915} C_VEL
LIN {X 0,Y 439.247,Z 386.125,A -85,B 0,C 180,E1 -15698.173,E2 -15698.173} C_VEL
LIN {X 0,Y 443.283,Z 356.55,A -85,B 0,C 180,E1 -15700.641,E2 -15700.641} C_VEL
LIN {X 0,Y 445.261,Z 356.47,A -85,B 0,C 180,E1 -15700.975,E2 -15700.975} C_VEL
LIN {X 0,Y 448.955,Z 354.156,A -85,B 0,C 180,E1 -15701.412,E2 -15701.412} C_VEL
LIN {X 0,Y 451.823,Z 351.613,A -85,B 0,C 180,E1 -15701.683,E2 -15701.683} C_VEL
LIN {X 0,Y 455.703,Z 349.897,A -85,B 0,C 180,E1 -15702.177,E2 -15702.177} C_VEL
LIN {X 0,Y 460.446,Z 346.36,A -85,B 0,C 180,E1 -15702.651,E2 -15702.651} C_VEL
LIN {X 0,Y 465.632,Z 343.618,A -85,B 0,C 180,E1 -15703.237,E2 -15703.237} C_VEL
LIN {X 0,Y 468.15,Z 341.884,A -85,B 0,C 180,E1 -15703.473,E2 -15703.473} C_VEL
LIN {X 0,Y 470.899,Z 349.839,A -85,B 0,C 180,E1 -15704.484,E2 -15704.484} C_VEL
LIN {X 0,Y 470.365,Z 372.226,A -85,B 0,C 180,E1 -15706.047,E2 -15706.047} C_VEL
LIN {X 0,Y 464.775,Z 398.05,A -85,B 0,C 180,E1 -15706.986,E2 -15706.986} C_VEL
LIN {X 0,Y 460.852,Z 480.196,A -85,B 0,C 180,E1 -15708.351,E2 -15708.351} C_VEL
LIN {X 0,Y 456.69,Z 542.095,A -85,B 0,C 180,E1 -15709.588,E2 -15709.588} C_VEL
LIN {X 0,Y 451.226,Z 607.78,A -85,B 0,C 180,E1 -15711.122,E2 -15711.122} C_VEL
LIN {X 0,Y 447.491,Z 653.023,A -85,B 0,C 180,E1 -15712.365,E2 -15712.365} C_VEL
LIN {X 0,Y 445.668,Z 677.543,A -85,B 0,C 180,E1 -15713.208,E2 -15713.208} C_VEL
LIN {X 0,Y 443.448,Z 699.052,A -85,B 0,C 180,E1 -15714.188,E2 -15714.188} C_VEL
LIN {X 0,Y 440.746,Z 719.67,A -85,B 0,C 180,E1 -15715.372,E2 -15715.372} C_VEL
LIN {X 0,Y 437.713,Z 739.284,A -85,B 0,C 180,E1 -15716.753,E2 -15716.753} C_VEL
LIN {X 0,Y 434.389,Z 758.036,A -85,B 0,C 180,E1 -15718.344,E2 -15718.344} C_VEL
LIN {X 0,Y 430.869,Z 775.879,A -85,B 0,C 180,E1 -15720.147,E2 -15720.147} C_VEL
LIN {X 0,Y 428.649,Z 786.403,A -85,B 0,C 180,E1 -15721.374,E2 -15721.374} C_VEL
LIN {X 0,Y 426.569,Z 792.199,A -85,B 0,C 180,E1 -15722.018,E2 -15722.018} C_VEL
LIN {X 0,Y 418.163,Z 806.503,A -85,B 0,C 180,E1 -15723.554,E2 -15723.554} C_VEL
LIN {X 0,Y 416.054,Z 811.677,A -85,B 0,C 180,E1 -15724.293,E2 -15724.293} C_VEL
LIN {X 0,Y 412.727,Z 825.579,A -85,B 0,C 180,E1 -15726.741,E2 -15726.741} C_VEL
LIN {X 0,Y 409.828,Z 837.724,A -85,B 0,C 180,E1 -15729.282,E2 -15729.282} C_VEL
LIN {X 0,Y 407.198,Z 848.973,A -85,B 0,C 180,E1 -15732.125,E2 -15732.125} C_VEL
LIN {X 0,Y 405.09,Z 858.595,A -85,B 0,C 180,E1 -15735.125,E2 -15735.125} C_VEL
LIN {X 0,Y 403.628,Z 865.866,A -85,B 0,C 180,E1 -15737.989,E2 -15737.989} C_VEL
LIN {X 0,Y 402.636,Z 871.479,A -85,B 0,C 180,E1 -15740.855,E2 -15740.855} C_VEL
LIN {X 0,Y 402.009,Z 875.701,A -85,B 0,C 180,E1 -15743.86,E2 -15743.86} C_VEL
LIN {X 0,Y 401.697,Z 878.215,A -85,B 0,C 180,E1 -15746.718,E2 -15746.718} C_VEL
LIN {X 0,Y 401.58,Z 879.177,A -85,B 0,C 180,E1 -15749.715,E2 -15749.715} C_VEL
LIN {X 0,Y 401.639,Z 878.588,A -85,B 0,C 180,E1 -15752.568,E2 -15752.568} C_VEL
LIN {X 0,Y 401.919,Z 876.416,A -85,B 0,C 180,E1 -15755.568,E2 -15755.568} C_VEL
LIN {X 0,Y 402.47,Z 872.618,A -85,B 0,C 180,E1 -15758.573,E2 -15758.573} C_VEL
LIN {X 0,Y 403.427,Z 867.074,A -85,B 0,C 180,E1 -15761.581,E2 -15761.581} C_VEL
LIN {X 0,Y 404.801,Z 859.988,A -85,B 0,C 180,E1 -15764.47,E2 -15764.47} C_VEL
LIN {X 0,Y 406.685,Z 851.263,A -85,B 0,C 180,E1 -15767.307,E2 -15767.307} C_VEL
LIN {X 0,Y 409.166,Z 840.507,A -85,B 0,C 180,E1 -15770.155,E2 -15770.155} C_VEL
LIN {X 0,Y 412.106,Z 828.21,A -85,B 0,C 180,E1 -15772.843,E2 -15772.843} C_VEL
LIN {X 0,Y 415.446,Z 814.375,A -85,B 0,C 180,E1 -15775.367,E2 -15775.367} C_VEL
LIN {X 0,Y 418.979,Z 799.456,A -85,B 0,C 180,E1 -15777.657,E2 -15777.657} C_VEL
LIN {X 0,Y 422.616,Z 783.429,A -85,B 0,C 180,E1 -15779.737,E2 -15779.737} C_VEL
LIN {X 0,Y 426.273,Z 766.208,A -85,B 0,C 180,E1 -15781.627,E2 -15781.627} C_VEL
LIN {X 0,Y 429.954,Z 747.171,A -85,B 0,C 180,E1 -15783.375,E2 -15783.375} C_VEL
LIN {X 0,Y 433.345,Z 727.035,A -85,B 0,C 180,E1 -15784.906,E2 -15784.906} C_VEL
LIN {X 0,Y 436.271,Z 706.649,A -85,B 0,C 180,E1 -15786.169,E2 -15786.169} C_VEL
LIN {X 0,Y 438.733,Z 685.135,A -85,B 0,C 180,E1 -15787.235,E2 -15787.235} C_VEL
LIN {X 0,Y 440.593,Z 663.377,A -85,B 0,C 180,E1 -15788.06,E2 -15788.06} C_VEL
LIN {X 0,Y 444.033,Z 620.387,A -85,B 0,C 180,E1 -15789.319,E2 -15789.319} C_VEL
LIN {X 0,Y 449.713,Z 556.319,A -85,B 0,C 180,E1 -15790.881,E2 -15790.881} C_VEL
LIN {X 0,Y 454.399,Z 491.907,A -85,B 0,C 180,E1 -15792.219,E2 -15792.219} C_VEL
LIN {X 0,Y 457.906,Z 425.096,A -85,B 0,C 180,E1 -15793.371,E2 -15793.371} C_VEL
LIN {X 0,Y 459.25,Z 398.805,A -85,B 0,C 180,E1 -15793.817,E2 -15793.817} C_VEL
LIN {X 0,Y 464.899,Z 373.15,A -85,B 0,C 180,E1 -15794.785,E2 -15794.785} C_VEL
LIN {X 0,Y 465.39,Z 353.946,A -85,B 0,C 180,E1 -15796.14,E2 -15796.14} C_VEL
LIN {X 0,Y 458.648,Z 335.098,A -85,B 0,C 180,E1 -15798.657,E2 -15798.657} C_VEL
LIN {X 0,Y 451.385,Z 317.254,A -85,B 0,C 180,E1 -15801.341,E2 -15801.341} C_VEL
LIN {X 0,Y 443.902,Z 301.367,A -85,B 0,C 180,E1 -15803.991,E2 -15803.991} C_VEL
LIN {X 0,Y 436.447,Z 287.134,A -85,B 0,C 180,E1 -15806.644,E2 -15806.644} C_VEL
LIN {X 0,Y 430.532,Z 276.878,A -85,B 0,C 180,E1 -15808.808,E2 -15808.808} C_VEL
LIN {X 0,Y 425.367,Z 268.39,A -85,B 0,C 180,E1 -15810.729,E2 -15810.729} C_VEL
LIN {X 0,Y 422.017,Z 263.167,A -85,B 0,C 180,E1 -15812.022,E2 -15812.022} C_VEL
LIN {X 0,Y 418.72,Z 258.143,A -85,B 0,C 180,E1 -15813.324,E2 -15813.324} C_VEL
LIN {X 0,Y 416.109,Z 254.486,A -85,B 0,C 180,E1 -15814.371,E2 -15814.371} C_VEL
LIN {X 0,Y 415.045,Z 252.734,A -85,B 0,C 180,E1 -15814.836,E2 -15814.836} C_VEL
LIN {X 0,Y 412.308,Z 249.235,A -85,B 0,C 180,E1 -15815.957,E2 -15815.957} C_VEL
LIN {X 0,Y 411.215,Z 247.12,A -85,B 0,C 180,E1 -15816.498,E2 -15816.498} C_VEL
LIN {X 0,Y 408.325,Z 244.044,A -85,B 0,C 180,E1 -15817.694,E2 -15817.694} C_VEL
LIN {X 0,Y 407.098,Z 241.256,A -85,B 0,C 180,E1 -15818.382,E2 -15818.382} C_VEL
LIN {X 0,Y 404.13,Z 238.776,A -85,B 0,C 180,E1 -15819.658,E2 -15819.658} C_VEL
LIN {X 0,Y 402.797,Z 235.839,A -85,B 0,C 180,E1 -15820.458,E2 -15820.458} C_VEL
LIN {X 0,Y 402.657,Z 235.03,A -85,B 0,C 180,E1 -15820.67,E2 -15820.67} C_VEL
LIN {X 0,Y 402.661,Z 235.068,A -85,B 0,C 180,E1 -15824.591,E2 -15824.591} C_VEL
LIN {X 0,Y 402.647,Z 235.02,A -85,B 0,C 180,E1 -15828.541,E2 -15828.541} C_VEL
LIN {X 0,Y 402.645,Z 235.035,A -85,B 0,C 180,E1 -15832.437,E2 -15832.437} C_VEL
LIN {X 0,Y 402.646,Z 235.058,A -85,B 0,C 180,E1 -15836.441,E2 -15836.441} C_VEL
LIN {X 0,Y 402.64,Z 235.014,A -85,B 0,C 180,E1 -15840.427,E2 -15840.427} C_VEL
LIN {X 0,Y 402.644,Z 235.069,A -85,B 0,C 180,E1 -15844.415,E2 -15844.415} C_VEL
LIN {X 0,Y 402.636,Z 235.025,A -85,B 0,C 180,E1 -15848.425,E2 -15848.425} C_VEL
LIN {X 0,Y 402.642,Z 235.077,A -85,B 0,C 180,E1 -15852.331,E2 -15852.331} C_VEL
LIN {X 0,Y 402.678,Z 235.295,A -85,B 0,C 180,E1 -15856.097,E2 -15856.097} C_VEL
LIN {X 0,Y 403.932,Z 238.535,A -85,B 0,C 180,E1 -15856.835,E2 -15856.835} C_VEL
LIN {X 0,Y 405.243,Z 240.418,A -85,B 0,C 180,E1 -15857.371,E2 -15857.371} C_VEL
LIN {X 0,Y 407.271,Z 244.299,A -85,B 0,C 180,E1 -15858.316,E2 -15858.316} C_VEL
LIN {X 0,Y 413.414,Z 256.133,A -85,B 0,C 180,E1 -15861.123,E2 -15861.123} C_VEL
LIN {X 0,Y 419.642,Z 267.863,A -85,B 0,C 180,E1 -15863.746,E2 -15863.746} C_VEL
LIN {X 0,Y 428.362,Z 284.928,A -85,B 0,C 180,E1 -15867.227,E2 -15867.227} C_VEL
LIN {X 0,Y 438.2,Z 304.91,A -85,B 0,C 180,E1 -15870.891,E2 -15870.891} C_VEL
LIN {X 0,Y 447.883,Z 325.197,A -85,B 0,C 180,E1 -15874.235,E2 -15874.235} C_VEL
LIN {X 0,Y 449.321,Z 327.855,A -85,B 0,C 180,E1 -15874.593,E2 -15874.593} C_VEL
LIN {X 0,Y 468.235,Z 357.336,A -85,B 0,C 180,E1 -15877.436,E2 -15877.436} C_VEL
LIN {X 0,Y 452.672,Z 602.957,A -85,B 0,C 180,E1 -15882.172,E2 -15882.172} C_VEL
LIN {X 0,Y 447.532,Z 693.393,A -85,B 0,C 180,E1 -15883.947,E2 -15883.947} C_VEL
LIN {X 0,Y 445.154,Z 717.934,A -85,B 0,C 180,E1 -15884.638,E2 -15884.638} C_VEL
LIN {X 0,Y 442.01,Z 743.924,A -85,B 0,C 180,E1 -15885.612,E2 -15885.612} C_VEL
LIN {X 0,Y 438.665,Z 767.287,A -85,B 0,C 180,E1 -15886.723,E2 -15886.723} C_VEL
LIN {X 0,Y 435.005,Z 789.351,A -85,B 0,C 180,E1 -15888.019,E2 -15888.019} C_VEL
LIN {X 0,Y 430.985,Z 811.601,A -85,B 0,C 180,E1 -15889.571,E2 -15889.571} C_VEL
LIN {X 0,Y 426.902,Z 832.266,A -85,B 0,C 180,E1 -15891.291,E2 -15891.291} C_VEL
LIN {X 0,Y 422.445,Z 853.607,A -85,B 0,C 180,E1 -15893.383,E2 -15893.383} C_VEL
LIN {X 0,Y 418.442,Z 872.322,A -85,B 0,C 180,E1 -15895.528,E2 -15895.528} C_VEL
LIN {X 0,Y 414.703,Z 889.344,A -85,B 0,C 180,E1 -15897.811,E2 -15897.811} C_VEL
LIN {X 0,Y 411.274,Z 905.352,A -85,B 0,C 180,E1 -15900.267,E2 -15900.267} C_VEL
LIN {X 0,Y 408.245,Z 919.956,A -85,B 0,C 180,E1 -15902.899,E2 -15902.899} C_VEL
LIN {X 0,Y 405.668,Z 933.438,A -85,B 0,C 180,E1 -15905.693,E2 -15905.693} C_VEL
LIN {X 0,Y 403.61,Z 945.51,A -85,B 0,C 180,E1 -15908.669,E2 -15908.669} C_VEL
LIN {X 0,Y 402.131,Z 956.233,A -85,B 0,C 180,E1 -15911.776,E2 -15911.776} C_VEL
LIN {X 0,Y 401.262,Z 964.473,A -85,B 0,C 180,E1 -15914.684,E2 -15914.684} C_VEL
LIN {X 0,Y 400.787,Z 971.664,A -85,B 0,C 180,E1 -15917.757,E2 -15917.757} C_VEL
LIN {X 0,Y 400.673,Z 977.063,A -85,B 0,C 180,E1 -15920.81,E2 -15920.81} C_VEL
LIN {X 0,Y 400.742,Z 980.667,A -85,B 0,C 180,E1 -15923.553,E2 -15923.553} C_VEL
LIN {X 0,Y 400.863,Z 983.322,A -85,B 0,C 180,E1 -15926.711,E2 -15926.711} C_VEL
LIN {X 0,Y 400.918,Z 984.21,A -85,B 0,C 180,E1 -15929.571,E2 -15929.571} C_VEL
LIN {X 0,Y 400.889,Z 983.899,A -85,B 0,C 180,E1 -15932.144,E2 -15932.144} C_VEL
LIN {X 0,Y 400.745,Z 982.323,A -85,B 0,C 180,E1 -15935.01,E2 -15935.01} C_VEL
LIN {X 0,Y 400.626,Z 979.002,A -85,B 0,C 180,E1 -15938.179,E2 -15938.179} C_VEL
LIN {X 0,Y 400.627,Z 974.586,A -85,B 0,C 180,E1 -15941.08,E2 -15941.08} C_VEL
LIN {X 0,Y 400.962,Z 968.262,A -85,B 0,C 180,E1 -15944.293,E2 -15944.293} C_VEL
LIN {X 0,Y 401.793,Z 960.095,A -85,B 0,C 180,E1 -15947.525,E2 -15947.525} C_VEL
LIN {X 0,Y 403.174,Z 950.792,A -85,B 0,C 180,E1 -15950.62,E2 -15950.62} C_VEL
LIN {X 0,Y 405.368,Z 939.105,A -85,B 0,C 180,E1 -15953.862,E2 -15953.862} C_VEL
LIN {X 0,Y 408.289,Z 926.172,A -85,B 0,C 180,E1 -15956.946,E2 -15956.946} C_VEL
LIN {X 0,Y 412.067,Z 911.092,A -85,B 0,C 180,E1 -15959.991,E2 -15959.991} C_VEL
LIN {X 0,Y 416.581,Z 894.718,A -85,B 0,C 180,E1 -15962.851,E2 -15962.851} C_VEL
LIN {X 0,Y 421.538,Z 877.5,A -85,B 0,C 180,E1 -15965.434,E2 -15965.434} C_VEL
LIN {X 0,Y 427.349,Z 857.778,A -85,B 0,C 180,E1 -15967.978,E2 -15967.978} C_VEL
LIN {X 0,Y 433.471,Z 837.335,A -85,B 0,C 180,E1 -15970.232,E2 -15970.232} C_VEL
LIN {X 0,Y 439.677,Z 816.077,A -85,B 0,C 180,E1 -15972.223,E2 -15972.223} C_VEL
LIN {X 0,Y 446.355,Z 792.602,A -85,B 0,C 180,E1 -15974.072,E2 -15974.072} C_VEL
LIN {X 0,Y 452.978,Z 768.224,A -85,B 0,C 180,E1 -15975.659,E2 -15975.659} C_VEL
LIN {X 0,Y 459.135,Z 744.038,A -85,B 0,C 180,E1 -15976.94,E2 -15976.94} C_VEL
LIN {X 0,Y 464.777,Z 719.677,A -85,B 0,C 180,E1 -15977.966,E2 -15977.966} C_VEL
LIN {X 0,Y 469.696,Z 695.435,A -85,B 0,C 180,E1 -15978.753,E2 -15978.753} C_VEL
LIN {X 0,Y 483.334,Z 618.38,A -85,B 0,C 180,E1 -15980.671,E2 -15980.671} C_VEL
LIN {X 0,Y 493.481,Z 571.567,A -85,B 0,C 180,E1 -15981.842,E2 -15981.842} C_VEL
LIN {X 0,Y 469.597,Z 672.835,A -85,B 0,C 180,E1 -15984.917,E2 -15984.917} C_VEL
LIN {X 0,Y 463.135,Z 699.906,A -85,B 0,C 180,E1 -15985.852,E2 -15985.852} C_VEL
LIN {X 0,Y 456.993,Z 722.138,A -85,B 0,C 180,E1 -15986.839,E2 -15986.839} C_VEL
LIN {X 0,Y 450.356,Z 744.439,A -85,B 0,C 180,E1 -15988.102,E2 -15988.102} C_VEL
LIN {X 0,Y 443.484,Z 766.764,A -85,B 0,C 180,E1 -15989.666,E2 -15989.666} C_VEL
LIN {X 0,Y 436.829,Z 788.198,A -85,B 0,C 180,E1 -15991.494,E2 -15991.494} C_VEL
LIN {X 0,Y 430.938,Z 807.473,A -85,B 0,C 180,E1 -15993.471,E2 -15993.471} C_VEL
LIN {X 0,Y 425.668,Z 824.709,A -85,B 0,C 180,E1 -15995.58,E2 -15995.58} C_VEL
LIN {X 0,Y 420.984,Z 839.947,A -85,B 0,C 180,E1 -15997.812,E2 -15997.812} C_VEL
LIN {X 0,Y 416.975,Z 852.881,A -85,B 0,C 180,E1 -16000.092,E2 -16000.092} C_VEL
LIN {X 0,Y 413.753,Z 863.124,A -85,B 0,C 180,E1 -16002.272,E2 -16002.272} C_VEL
LIN {X 0,Y 410.689,Z 872.523,A -85,B 0,C 180,E1 -16004.755,E2 -16004.755} C_VEL
LIN {X 0,Y 408.052,Z 880.19,A -85,B 0,C 180,E1 -16007.403,E2 -16007.403} C_VEL
LIN {X 0,Y 405.987,Z 885.686,A -85,B 0,C 180,E1 -16010.073,E2 -16010.073} C_VEL
LIN {X 0,Y 404.518,Z 889.004,A -85,B 0,C 180,E1 -16012.615,E2 -16012.615} C_VEL
LIN {X 0,Y 403.429,Z 890.534,A -85,B 0,C 180,E1 -16015.166,E2 -16015.166} C_VEL
LIN {X 0,Y 402.684,Z 890.319,A -85,B 0,C 180,E1 -16017.723,E2 -16017.723} C_VEL
LIN {X 0,Y 402.235,Z 888.345,A -85,B 0,C 180,E1 -16020.285,E2 -16020.285} C_VEL
LIN {X 0,Y 402.024,Z 884.497,A -85,B 0,C 180,E1 -16022.933,E2 -16022.933} C_VEL
LIN {X 0,Y 402.075,Z 878.77,A -85,B 0,C 180,E1 -16025.566,E2 -16025.566} C_VEL
LIN {X 0,Y 402.387,Z 871.247,A -85,B 0,C 180,E1 -16028.143,E2 -16028.143} C_VEL
LIN {X 0,Y 402.97,Z 862.228,A -85,B 0,C 180,E1 -16030.581,E2 -16030.581} C_VEL
LIN {X 0,Y 403.897,Z 851.146,A -85,B 0,C 180,E1 -16033.019,E2 -16033.019} C_VEL
LIN {X 0,Y 405.115,Z 838.563,A -85,B 0,C 180,E1 -16035.313,E2 -16035.313} C_VEL
LIN {X 0,Y 406.656,Z 824.022,A -85,B 0,C 180,E1 -16037.53,E2 -16037.53} C_VEL
LIN {X 0,Y 408.451,Z 807.884,A -85,B 0,C 180,E1 -16039.596,E2 -16039.596} C_VEL
LIN {X 0,Y 410.452,Z 790.07,A -85,B 0,C 180,E1 -16041.5,E2 -16041.5} C_VEL
LIN {X 0,Y 412.515,Z 770.976,A -85,B 0,C 180,E1 -16043.196,E2 -16043.196} C_VEL
LIN {X 0,Y 414.606,Z 751.017,A -85,B 0,C 180,E1 -16044.659,E2 -16044.659} C_VEL
LIN {X 0,Y 416.732,Z 728.916,A -85,B 0,C 180,E1 -16045.969,E2 -16045.969} C_VEL
LIN {X 0,Y 418.597,Z 706.926,A -85,B 0,C 180,E1 -16046.991,E2 -16046.991} C_VEL
LIN {X 0,Y 420.286,Z 683.864,A -85,B 0,C 180,E1 -16047.79,E2 -16047.79} C_VEL
LIN {X 0,Y 430.531,Z 507.577,A -85,B 0,C 180,E1 -16052.057,E2 -16052.057} C_VEL
LIN {X 0,Y 425.719,Z 436.95,A -85,B 0,C 180,E1 -16054.475,E2 -16054.475} C_VEL
LIN {X 0,Y 432.556,Z 384.765,A -85,B 0,C 180,E1 -16058.865,E2 -16058.865} C_VEL
LIN {X 0,Y 434.747,Z 369.445,A -85,B 0,C 180,E1 -16060.176,E2 -16060.176} C_VEL
LIN {X 0,Y 436.878,Z 369.238,A -85,B 0,C 180,E1 -16060.542,E2 -16060.542} C_VEL
LIN {X 0,Y 440.571,Z 366.73,A -85,B 0,C 180,E1 -16060.988,E2 -16060.988} C_VEL
LIN {X 0,Y 443.446,Z 363.976,A -85,B 0,C 180,E1 -16061.265,E2 -16061.265} C_VEL
LIN {X 0,Y 447.29,Z 362.213,A -85,B 0,C 180,E1 -16061.772,E2 -16061.772} C_VEL
LIN {X 0,Y 452.013,Z 358.506,A -85,B 0,C 180,E1 -16062.259,E2 -16062.259} C_VEL
LIN {X 0,Y 457.127,Z 355.759,A -85,B 0,C 180,E1 -16062.864,E2 -16062.864} C_VEL
LIN {X 0,Y 461.074,Z 352.937,A -85,B 0,C 180,E1 -16063.258,E2 -16063.258} C_VEL
LIN {X 0,Y 464.419,Z 351.348,A -85,B 0,C 180,E1 -16063.642,E2 -16063.642} C_VEL
LIN {X 0,Y 465.273,Z 353.834,A -85,B 0,C 180,E1 -16063.959,E2 -16063.959} C_VEL
LIN {X 0,Y 464.706,Z 374.053,A -85,B 0,C 180,E1 -16065.37,E2 -16065.37} C_VEL
LIN {X 0,Y 458.913,Z 400.652,A -85,B 0,C 180,E1 -16066.335,E2 -16066.335} C_VEL
LIN {X 0,Y 454.883,Z 482.443,A -85,B 0,C 180,E1 -16067.706,E2 -16067.706} C_VEL
LIN {X 0,Y 450.628,Z 543.813,A -85,B 0,C 180,E1 -16068.944,E2 -16068.944} C_VEL
LIN {X 0,Y 445.098,Z 608.261,A -85,B 0,C 180,E1 -16070.467,E2 -16070.467} C_VEL
LIN {X 0,Y 441.209,Z 653.482,A -85,B 0,C 180,E1 -16071.728,E2 -16071.728} C_VEL
LIN {X 0,Y 439.257,Z 678.779,A -85,B 0,C 180,E1 -16072.608,E2 -16072.608} C_VEL
LIN {X 0,Y 437.018,Z 699.883,A -85,B 0,C 180,E1 -16073.578,E2 -16073.578} C_VEL
LIN {X 0,Y 434.264,Z 720.371,A -85,B 0,C 180,E1 -16074.761,E2 -16074.761} C_VEL
LIN {X 0,Y 431.083,Z 740.248,A -85,B 0,C 180,E1 -16076.174,E2 -16076.174} C_VEL
LIN {X 0,Y 427.636,Z 759.025,A -85,B 0,C 180,E1 -16077.784,E2 -16077.784} C_VEL
LIN {X 0,Y 423.984,Z 776.893,A -85,B 0,C 180,E1 -16079.611,E2 -16079.611} C_VEL
LIN {X 0,Y 420.21,Z 793.987,A -85,B 0,C 180,E1 -16081.693,E2 -16081.693} C_VEL
LIN {X 0,Y 416.587,Z 809.547,A -85,B 0,C 180,E1 -16083.945,E2 -16083.945} C_VEL
LIN {X 0,Y 416.054,Z 811.677,A -85,B 0,C 180,E1 -16084.293,E2 -16084.293} C_VEL
LIN {X 0,Y 413.964,Z 816.792,A -85,B 0,C 180,E1 -16085.058,E2 -16085.058} C_VEL
LIN {X 0,Y 405.606,Z 829.339,A -85,B 0,C 180,E1 -16086.913,E2 -16086.913} C_VEL
LIN {X 0,Y 403.593,Z 833.764,A -85,B 0,C 180,E1 -16087.769,E2 -16087.769} C_VEL
LIN {X 0,Y 400.764,Z 845.186,A -85,B 0,C 180,E1 -16090.468,E2 -16090.468} C_VEL
LIN {X 0,Y 398.356,Z 855.299,A -85,B 0,C 180,E1 -16093.373,E2 -16093.373} C_VEL
LIN {X 0,Y 396.472,Z 863.836,A -85,B 0,C 180,E1 -16096.435,E2 -16096.435} C_VEL
LIN {X 0,Y 395.142,Z 870.452,A -85,B 0,C 180,E1 -16099.502,E2 -16099.502} C_VEL
LIN {X 0,Y 394.317,Z 875.294,A -85,B 0,C 180,E1 -16102.569,E2 -16102.569} C_VEL
LIN {X 0,Y 393.853,Z 878.467,A -85,B 0,C 180,E1 -16105.632,E2 -16105.632} C_VEL
LIN {X 0,Y 393.662,Z 880.005,A -85,B 0,C 180,E1 -16108.544,E2 -16108.544} C_VEL
LIN {X 0,Y 393.658,Z 880.02,A -85,B 0,C 180,E1 -16111.455,E2 -16111.455} C_VEL
LIN {X 0,Y 393.845,Z 878.542,A -85,B 0,C 180,E1 -16114.368,E2 -16114.368} C_VEL
LIN {X 0,Y 394.311,Z 875.372,A -85,B 0,C 180,E1 -16117.476,E2 -16117.476} C_VEL
LIN {X 0,Y 395.114,Z 870.659,A -85,B 0,C 180,E1 -16120.498,E2 -16120.498} C_VEL
LIN {X 0,Y 396.436,Z 864.108,A -85,B 0,C 180,E1 -16123.566,E2 -16123.566} C_VEL
LIN {X 0,Y 398.3,Z 855.618,A -85,B 0,C 180,E1 -16126.63,E2 -16126.63} C_VEL
LIN {X 0,Y 400.692,Z 845.567,A -85,B 0,C 180,E1 -16129.535,E2 -16129.535} C_VEL
LIN {X 0,Y 403.555,Z 834.031,A -85,B 0,C 180,E1 -16132.277,E2 -16132.277} C_VEL
LIN {X 0,Y 406.827,Z 821.049,A -85,B 0,C 180,E1 -16134.852,E2 -16134.852} C_VEL
LIN {X 0,Y 410.422,Z 806.621,A -85,B 0,C 180,E1 -16137.259,E2 -16137.259} C_VEL
LIN {X 0,Y 414.255,Z 790.673,A -85,B 0,C 180,E1 -16139.498,E2 -16139.498} C_VEL
LIN {X 0,Y 418.229,Z 773.076,A -85,B 0,C 180,E1 -16141.573,E2 -16141.573} C_VEL
LIN {X 0,Y 421.949,Z 755.104,A -85,B 0,C 180,E1 -16143.351,E2 -16143.351} C_VEL
LIN {X 0,Y 425.438,Z 736.261,A -85,B 0,C 180,E1 -16144.91,E2 -16144.91} C_VEL
LIN {X 0,Y 428.589,Z 716.572,A -85,B 0,C 180,E1 -16146.257,E2 -16146.257} C_VEL
LIN {X 0,Y 431.311,Z 695.996,A -85,B 0,C 180,E1 -16147.401,E2 -16147.401} C_VEL
LIN {X 0,Y 433.518,Z 674.401,A -85,B 0,C 180,E1 -16148.343,E2 -16148.343} C_VEL
LIN {X 0,Y 436.584,Z 635.577,A -85,B 0,C 180,E1 -16149.583,E2 -16149.583} C_VEL
LIN {X 0,Y 442.217,Z 574.88,A -85,B 0,C 180,E1 -16151.146,E2 -16151.146} C_VEL
LIN {X 0,Y 447.096,Z 514.41,A -85,B 0,C 180,E1 -16152.479,E2 -16152.479} C_VEL
LIN {X 0,Y 450.829,Z 453.05,A -85,B 0,C 180,E1 -16153.617,E2 -16153.617} C_VEL
LIN {X 0,Y 453.44,Z 401.597,A -85,B 0,C 180,E1 -16154.481,E2 -16154.481} C_VEL
LIN {X 0,Y 459.348,Z 375.023,A -85,B 0,C 180,E1 -16155.47,E2 -16155.47} C_VEL
LIN {X 0,Y 459.819,Z 357.957,A -85,B 0,C 180,E1 -16156.68,E2 -16156.68} C_VEL
LIN {X 0,Y 453.126,Z 339.263,A -85,B 0,C 180,E1 -16159.219,E2 -16159.219} C_VEL
LIN {X 0,Y 445.964,Z 321.559,A -85,B 0,C 180,E1 -16161.933,E2 -16161.933} C_VEL
LIN {X 0,Y 438.631,Z 305.81,A -85,B 0,C 180,E1 -16164.619,E2 -16164.619} C_VEL
LIN {X 0,Y 430.985,Z 291.238,A -85,B 0,C 180,E1 -16167.436,E2 -16167.436} C_VEL
LIN {X 0,Y 424.483,Z 279.873,A -85,B 0,C 180,E1 -16169.885,E2 -16169.885} C_VEL
LIN {X 0,Y 418.521,Z 270.199,A -85,B 0,C 180,E1 -16172.233,E2 -16172.233} C_VEL
LIN {X 0,Y 414.86,Z 264.72,A -85,B 0,C 180,E1 -16173.713,E2 -16173.713} C_VEL
LIN {X 0,Y 411.559,Z 259.659,A -85,B 0,C 180,E1 -16175.146,E2 -16175.146} C_VEL
LIN {X 0,Y 408.684,Z 255.692,A -85,B 0,C 180,E1 -16176.382,E2 -16176.382} C_VEL
LIN {X 0,Y 407.759,Z 254.125,A -85,B 0,C 180,E1 -16176.823,E2 -16176.823} C_VEL
LIN {X 0,Y 404.939,Z 250.788,A -85,B 0,C 180,E1 -16178.07,E2 -16178.07} C_VEL
LIN {X 0,Y 403.917,Z 248.503,A -85,B 0,C 180,E1 -16178.66,E2 -16178.66} C_VEL
LIN {X 0,Y 401.052,Z 245.867,A -85,B 0,C 180,E1 -16179.952,E2 -16179.952} C_VEL
LIN {X 0,Y 399.313,Z 242.292,A -85,B 0,C 180,E1 -16181.003,E2 -16181.003} C_VEL
LIN {X 0,Y 396.223,Z 239.78,A -85,B 0,C 180,E1 -16182.524,E2 -16182.524} C_VEL
LIN {X 0,Y 394.845,Z 236.765,A -85,B 0,C 180,E1 -16183.496,E2 -16183.496} C_VEL
LIN {X 0,Y 394.719,Z 236.027,A -85,B 0,C 180,E1 -16183.669,E2 -16183.669} C_VEL
LIN {X 0,Y 394.715,Z 236.003,A -85,B 0,C 180,E1 -16187.566,E2 -16187.566} C_VEL
LIN {X 0,Y 394.724,Z 236.047,A -85,B 0,C 180,E1 -16191.551,E2 -16191.551} C_VEL
LIN {X 0,Y 394.716,Z 236.016,A -85,B 0,C 180,E1 -16195.496,E2 -16195.496} C_VEL
LIN {X 0,Y 394.72,Z 236.009,A -85,B 0,C 180,E1 -16199.419,E2 -16199.419} C_VEL
LIN {X 0,Y 394.723,Z 236.06,A -85,B 0,C 180,E1 -16203.485,E2 -16203.485} C_VEL
LIN {X 0,Y 394.725,Z 235.999,A -85,B 0,C 180,E1 -16207.569,E2 -16207.569} C_VEL
LIN {X 0,Y 394.725,Z 236.06,A -85,B 0,C 180,E1 -16211.544,E2 -16211.544} C_VEL
LIN {X 0,Y 394.723,Z 236.223,A -85,B 0,C 180,E1 -16214.561,E2 -16214.561} C_VEL
LIN {X 0,Y 396.103,Z 239.627,A -85,B 0,C 180,E1 -16215.37,E2 -16215.37} C_VEL
LIN {X 0,Y 397.354,Z 241.451,A -85,B 0,C 180,E1 -16215.919,E2 -16215.919} C_VEL
LIN {X 0,Y 399.276,Z 245.225,A -85,B 0,C 180,E1 -16216.888,E2 -16216.888} C_VEL
LIN {X 0,Y 404.844,Z 255.697,A -85,B 0,C 180,E1 -16219.477,E2 -16219.477} C_VEL
LIN {X 0,Y 412.442,Z 270.324,A -85,B 0,C 180,E1 -16222.823,E2 -16222.823} C_VEL
LIN {X 0,Y 420.762,Z 286.51,A -85,B 0,C 180,E1 -16226.232,E2 -16226.232} C_VEL
LIN {X 0,Y 430.872,Z 306.895,A -85,B 0,C 180,E1 -16230.083,E2 -16230.083} C_VEL
LIN {X 0,Y 441.101,Z 328.179,A -85,B 0,C 180,E1 -16233.658,E2 -16233.658} C_VEL
LIN {X 0,Y 461.877,Z 360.637,A -85,B 0,C 180,E1 -16236.863,E2 -16236.863} C_VEL
LIN {X 0,Y 445.47,Z 611.489,A -85,B 0,C 180,E1 -16241.782,E2 -16241.782} C_VEL
LIN {X 0,Y 440.619,Z 693.447,A -85,B 0,C 180,E1 -16243.428,E2 -16243.428} C_VEL
LIN {X 0,Y 438.181,Z 717.872,A -85,B 0,C 180,E1 -16244.129,E2 -16244.129} C_VEL
LIN {X 0,Y 434.969,Z 743.728,A -85,B 0,C 180,E1 -16245.112,E2 -16245.112} C_VEL
LIN {X 0,Y 431.633,Z 766.481,A -85,B 0,C 180,E1 -16246.206,E2 -16246.206} C_VEL
LIN {X 0,Y 427.886,Z 788.627,A -85,B 0,C 180,E1 -16247.52,E2 -16247.52} C_VEL
LIN {X 0,Y 423.763,Z 810.906,A -85,B 0,C 180,E1 -16249.092,E2 -16249.092} C_VEL
LIN {X 0,Y 419.579,Z 831.575,A -85,B 0,C 180,E1 -16250.838,E2 -16250.838} C_VEL
LIN {X 0,Y 415.003,Z 852.964,A -85,B 0,C 180,E1 -16252.962,E2 -16252.962} C_VEL
LIN {X 0,Y 410.924,Z 871.57,A -85,B 0,C 180,E1 -16255.123,E2 -16255.123} C_VEL
LIN {X 0,Y 406.955,Z 889.233,A -85,B 0,C 180,E1 -16257.53,E2 -16257.53} C_VEL
LIN {X 0,Y 403.342,Z 905.635,A -85,B 0,C 180,E1 -16260.114,E2 -16260.114} C_VEL
LIN {X 0,Y 400.265,Z 920.149,A -85,B 0,C 180,E1 -16262.797,E2 -16262.797} C_VEL
LIN {X 0,Y 397.541,Z 934.122,A -85,B 0,C 180,E1 -16265.797,E2 -16265.797} C_VEL
LIN {X 0,Y 395.598,Z 945.41,A -85,B 0,C 180,E1 -16268.656,E2 -16268.656} C_VEL
LIN {X 0,Y 394.063,Z 956.397,A -85,B 0,C 180,E1 -16271.967,E2 -16271.967} C_VEL
LIN {X 0,Y 393.258,Z 964.212,A -85,B 0,C 180,E1 -16274.818,E2 -16274.818} C_VEL
LIN {X 0,Y 392.785,Z 971.796,A -85,B 0,C 180,E1 -16278.25,E2 -16278.25} C_VEL
LIN {X 0,Y 392.716,Z 976.546,A -85,B 0,C 180,E1 -16281.073,E2 -16281.073} C_VEL
LIN {X 0,Y 392.812,Z 980.195,A -85,B 0,C 180,E1 -16284.01,E2 -16284.01} C_VEL
LIN {X 0,Y 392.931,Z 982.478,A -85,B 0,C 180,E1 -16287.083,E2 -16287.083} C_VEL
LIN {X 0,Y 392.993,Z 983.233,A -85,B 0,C 180,E1 -16289.854,E2 -16289.854} C_VEL
LIN {X 0,Y 392.923,Z 982.838,A -85,B 0,C 180,E1 -16292.48,E2 -16292.48} C_VEL
LIN {X 0,Y 392.774,Z 981.073,A -85,B 0,C 180,E1 -16295.551,E2 -16295.551} C_VEL
LIN {X 0,Y 392.632,Z 977.508,A -85,B 0,C 180,E1 -16298.789,E2 -16298.789} C_VEL
LIN {X 0,Y 392.68,Z 972.943,A -85,B 0,C 180,E1 -16301.754,E2 -16301.754} C_VEL
LIN {X 0,Y 393.149,Z 966.031,A -85,B 0,C 180,E1 -16305.186,E2 -16305.186} C_VEL
LIN {X 0,Y 394.093,Z 958.065,A -85,B 0,C 180,E1 -16308.338,E2 -16308.338} C_VEL
LIN {X 0,Y 395.854,Z 947.573,A -85,B 0,C 180,E1 -16311.796,E2 -16311.796} C_VEL
LIN {X 0,Y 398.258,Z 936.146,A -85,B 0,C 180,E1 -16314.948,E2 -16314.948} C_VEL
LIN {X 0,Y 401.89,Z 921.536,A -85,B 0,C 180,E1 -16318.373,E2 -16318.373} C_VEL
LIN {X 0,Y 405.979,Z 906.89,A -85,B 0,C 180,E1 -16321.311,E2 -16321.311} C_VEL
LIN {X 0,Y 410.944,Z 890.086,A -85,B 0,C 180,E1 -16324.198,E2 -16324.198} C_VEL
LIN {X 0,Y 416.595,Z 872.055,A -85,B 0,C 180,E1 -16326.873,E2 -16326.873} C_VEL
LIN {X 0,Y 422.605,Z 853.132,A -85,B 0,C 180,E1 -16329.265,E2 -16329.265} C_VEL
LIN {X 0,Y 429.388,Z 831.772,A -85,B 0,C 180,E1 -16331.58,E2 -16331.58} C_VEL
LIN {X 0,Y 436.361,Z 809.637,A -85,B 0,C 180,E1 -16333.608,E2 -16333.608} C_VEL
LIN {X 0,Y 443.373,Z 786.731,A -85,B 0,C 180,E1 -16335.358,E2 -16335.358} C_VEL
LIN {X 0,Y 450.057,Z 763.599,A -85,B 0,C 180,E1 -16336.82,E2 -16336.82} C_VEL
LIN {X 0,Y 456.498,Z 739.939,A -85,B 0,C 180,E1 -16338.041,E2 -16338.041} C_VEL
LIN {X 0,Y 462.208,Z 717.359,A -85,B 0,C 180,E1 -16338.977,E2 -16338.977} C_VEL
LIN {X 0,Y 467.629,Z 692.711,A -85,B 0,C 180,E1 -16339.766,E2 -16339.766} C_VEL
LIN {X 0,Y 481.281,Z 623.058,A -85,B 0,C 180,E1 -16341.511,E2 -16341.511} C_VEL
LIN {X 0,Y 484.763,Z 607.39,A -85,B 0,C 180,E1 -16341.916,E2 -16341.916} C_VEL
LIN {X 0,Y 463.628,Z 693.211,A -85,B 0,C 180,E1 -16344.596,E2 -16344.596} C_VEL
LIN {X 0,Y 456.879,Z 716.529,A -85,B 0,C 180,E1 -16345.547,E2 -16345.547} C_VEL
LIN {X 0,Y 449.865,Z 738.42,A -85,B 0,C 180,E1 -16346.702,E2 -16346.702} C_VEL
LIN {X 0,Y 442.192,Z 761.052,A -85,B 0,C 180,E1 -16348.206,E2 -16348.206} C_VEL
LIN {X 0,Y 434.461,Z 783.348,A -85,B 0,C 180,E1 -16350.039,E2 -16350.039} C_VEL
LIN {X 0,Y 427.57,Z 803.392,A -85,B 0,C 180,E1 -16352.038,E2 -16352.038} C_VEL
LIN {X 0,Y 421.307,Z 821.917,A -85,B 0,C 180,E1 -16354.258,E2 -16354.258} C_VEL
LIN {X 0,Y 416.071,Z 837.49,A -85,B 0,C 180,E1 -16356.489,E2 -16356.489} C_VEL
LIN {X 0,Y 411.566,Z 850.821,A -85,B 0,C 180,E1 -16358.777,E2 -16358.777} C_VEL
LIN {X 0,Y 407.505,Z 862.67,A -85,B 0,C 180,E1 -16361.25,E2 -16361.25} C_VEL
LIN {X 0,Y 404.257,Z 871.817,A -85,B 0,C 180,E1 -16363.622,E2 -16363.622} C_VEL
LIN {X 0,Y 401.41,Z 879.548,A -85,B 0,C 180,E1 -16366.165,E2 -16366.165} C_VEL
LIN {X 0,Y 399.007,Z 885.589,A -85,B 0,C 180,E1 -16368.874,E2 -16368.874} C_VEL
LIN {X 0,Y 397.256,Z 889.417,A -85,B 0,C 180,E1 -16371.46,E2 -16371.46} C_VEL
LIN {X 0,Y 396.023,Z 891.442,A -85,B 0,C 180,E1 -16373.913,E2 -16373.913} C_VEL
LIN {X 0,Y 395.082,Z 891.845,A -85,B 0,C 180,E1 -16376.518,E2 -16376.518} C_VEL
LIN {X 0,Y 394.473,Z 890.47,A -85,B 0,C 180,E1 -16379.129,E2 -16379.129} C_VEL
LIN {X 0,Y 394.138,Z 887.359,A -85,B 0,C 180,E1 -16381.745,E2 -16381.745} C_VEL
LIN {X 0,Y 394.06,Z 882.487,A -85,B 0,C 180,E1 -16384.366,E2 -16384.366} C_VEL
LIN {X 0,Y 394.256,Z 875.77,A -85,B 0,C 180,E1 -16386.992,E2 -16386.992} C_VEL
LIN {X 0,Y 394.704,Z 867.579,A -85,B 0,C 180,E1 -16389.478,E2 -16389.478} C_VEL
LIN {X 0,Y 395.478,Z 857.425,A -85,B 0,C 180,E1 -16391.966,E2 -16391.966} C_VEL
LIN {X 0,Y 396.553,Z 845.844,A -85,B 0,C 180,E1 -16394.306,E2 -16394.306} C_VEL
LIN {X 0,Y 397.993,Z 831.999,A -85,B 0,C 180,E1 -16396.643,E2 -16396.643} C_VEL
LIN {X 0,Y 399.72,Z 816.558,A -85,B 0,C 180,E1 -16398.826,E2 -16398.826} C_VEL
LIN {X 0,Y 401.687,Z 799.484,A -85,B 0,C 180,E1 -16400.852,E2 -16400.852} C_VEL
LIN {X 0,Y 403.836,Z 780.552,A -85,B 0,C 180,E1 -16402.722,E2 -16402.722} C_VEL
LIN {X 0,Y 405.964,Z 761.165,A -85,B 0,C 180,E1 -16404.312,E2 -16404.312} C_VEL
LIN {X 0,Y 408.237,Z 739.392,A -85,B 0,C 180,E1 -16405.769,E2 -16405.769} C_VEL
LIN {X 0,Y 410.237,Z 717.786,A -85,B 0,C 180,E1 -16406.92,E2 -16406.92} C_VEL
LIN {X 0,Y 412.11,Z 694.835,A -85,B 0,C 180,E1 -16407.858,E2 -16407.858} C_VEL
LIN {X 0,Y 413.709,Z 669.985,A -85,B 0,C 180,E1 -16408.576,E2 -16408.576} C_VEL
LIN {X 0,Y 423.42,Z 508.339,A -85,B 0,C 180,E1 -16412.545,E2 -16412.545} C_VEL
LIN {X 0,Y 418.715,Z 436.254,A -85,B 0,C 180,E1 -16415.066,E2 -16415.066} C_VEL
LIN {X 0,Y 425.681,Z 384.922,A -85,B 0,C 180,E1 -16419.44,E2 -16419.44} C_VEL
LIN {X 0,Y 426.131,Z 382.75,A -85,B 0,C 180,E1 -16419.66,E2 -16419.66} C_VEL
LIN {X 0,Y 427.915,Z 382.591,A -85,B 0,C 180,E1 -16419.985,E2 -16419.985} C_VEL
LIN {X 0,Y 431.503,Z 380.197,A -85,B 0,C 180,E1 -16420.453,E2 -16420.453} C_VEL
LIN {X 0,Y 434.781,Z 376.908,A -85,B 0,C 180,E1 -16420.778,E2 -16420.778} C_VEL
LIN {X 0,Y 438.189,Z 375.386,A -85,B 0,C 180,E1 -16421.259,E2 -16421.259} C_VEL
LIN {X 0,Y 442.82,Z 371.714,A -85,B 0,C 180,E1 -16421.768,E2 -16421.768} C_VEL
LIN {X 0,Y 444.353,Z 370.603,A -85,B 0,C 180,E1 -16421.937,E2 -16421.937} C_VEL
LIN {X 0,Y 449.493,Z 367.543,A -85,B 0,C 180,E1 -16422.551,E2 -16422.551} C_VEL
LIN {X 0,Y 452.639,Z 365.106,A -85,B 0,C 180,E1 -16422.874,E2 -16422.874} C_VEL
LIN {X 0,Y 458.648,Z 361.576,A -85,B 0,C 180,E1 -16423.544,E2 -16423.544} C_VEL
LIN {X 0,Y 459.587,Z 361.052,A -85,B 0,C 180,E1 -16423.648,E2 -16423.648} C_VEL
LIN {X 0,Y 459.113,Z 375.887,A -85,B 0,C 180,E1 -16424.677,E2 -16424.677} C_VEL
LIN {X 0,Y 453.096,Z 403.543,A -85,B 0,C 180,E1 -16425.672,E2 -16425.672} C_VEL
LIN {X 0,Y 448.959,Z 484.898,A -85,B 0,C 180,E1 -16427.047,E2 -16427.047} C_VEL
LIN {X 0,Y 444.604,Z 545.798,A -85,B 0,C 180,E1 -16428.289,E2 -16428.289} C_VEL
LIN {X 0,Y 438.973,Z 609.349,A -85,B 0,C 180,E1 -16429.81,E2 -16429.81} C_VEL
LIN {X 0,Y 434.943,Z 654.494,A -85,B 0,C 180,E1 -16431.09,E2 -16431.09} C_VEL
LIN {X 0,Y 432.878,Z 680.322,A -85,B 0,C 180,E1 -16432,E2 -16432} C_VEL
LIN {X 0,Y 430.481,Z 702.025,A -85,B 0,C 180,E1 -16433.016,E2 -16433.016} C_VEL
LIN {X 0,Y 427.457,Z 723.411,A -85,B 0,C 180,E1 -16434.286,E2 -16434.286} C_VEL
LIN {X 0,Y 424.019,Z 743.836,A -85,B 0,C 180,E1 -16435.789,E2 -16435.789} C_VEL
LIN {X 0,Y 420.34,Z 762.822,A -85,B 0,C 180,E1 -16437.479,E2 -16437.479} C_VEL
LIN {X 0,Y 416.453,Z 780.856,A -85,B 0,C 180,E1 -16439.402,E2 -16439.402} C_VEL
LIN {X 0,Y 412.647,Z 797.284,A -85,B 0,C 180,E1 -16441.487,E2 -16441.487} C_VEL
LIN {X 0,Y 408.993,Z 812.278,A -85,B 0,C 180,E1 -16443.736,E2 -16443.736} C_VEL
LIN {X 0,Y 405.404,Z 826.606,A -85,B 0,C 180,E1 -16446.295,E2 -16446.295} C_VEL
LIN {X 0,Y 403.593,Z 833.764,A -85,B 0,C 180,E1 -16447.769,E2 -16447.769} C_VEL
LIN {X 0,Y 401.613,Z 838.098,A -85,B 0,C 180,E1 -16448.65,E2 -16448.65} C_VEL
LIN {X 0,Y 393.52,Z 848.674,A -85,B 0,C 180,E1 -16450.82,E2 -16450.82} C_VEL
LIN {X 0,Y 391.69,Z 852.277,A -85,B 0,C 180,E1 -16451.788,E2 -16451.788} C_VEL
LIN {X 0,Y 389.483,Z 861.436,A -85,B 0,C 180,E1 -16454.82,E2 -16454.82} C_VEL
LIN {X 0,Y 387.84,Z 868.881,A -85,B 0,C 180,E1 -16457.946,E2 -16457.946} C_VEL
LIN {X 0,Y 386.745,Z 874.456,A -85,B 0,C 180,E1 -16461.076,E2 -16461.076} C_VEL
LIN {X 0,Y 386.124,Z 878.167,A -85,B 0,C 180,E1 -16464.054,E2 -16464.054} C_VEL
LIN {X 0,Y 385.79,Z 880.481,A -85,B 0,C 180,E1 -16467.177,E2 -16467.177} C_VEL
LIN {X 0,Y 385.713,Z 881.216,A -85,B 0,C 180,E1 -16470.148,E2 -16470.148} C_VEL
LIN {X 0,Y 385.816,Z 880.333,A -85,B 0,C 180,E1 -16473.268,E2 -16473.268} C_VEL
LIN {X 0,Y 386.158,Z 877.967,A -85,B 0,C 180,E1 -16476.243,E2 -16476.243} C_VEL
LIN {X 0,Y 386.888,Z 873.665,A -85,B 0,C 180,E1 -16479.521,E2 -16479.521} C_VEL
LIN {X 0,Y 388.069,Z 867.79,A -85,B 0,C 180,E1 -16482.651,E2 -16482.651} C_VEL
LIN {X 0,Y 389.714,Z 860.493,A -85,B 0,C 180,E1 -16485.628,E2 -16485.628} C_VEL
LIN {X 0,Y 391.951,Z 851.375,A -85,B 0,C 180,E1 -16488.595,E2 -16488.595} C_VEL
LIN {X 0,Y 394.838,Z 840.203,A -85,B 0,C 180,E1 -16491.543,E2 -16491.543} C_VEL
LIN {X 0,Y 398.208,Z 827.425,A -85,B 0,C 180,E1 -16494.318,E2 -16494.318} C_VEL
LIN {X 0,Y 401.975,Z 813.051,A -85,B 0,C 180,E1 -16496.918,E2 -16496.918} C_VEL
LIN {X 0,Y 405.796,Z 798.001,A -85,B 0,C 180,E1 -16499.201,E2 -16499.201} C_VEL
LIN {X 0,Y 409.769,Z 781.494,A -85,B 0,C 180,E1 -16501.315,E2 -16501.315} C_VEL
LIN {X 0,Y 413.668,Z 764.057,A -85,B 0,C 180,E1 -16503.194,E2 -16503.194} C_VEL
LIN {X 0,Y 417.35,Z 745.801,A -85,B 0,C 180,E1 -16504.848,E2 -16504.848} C_VEL
LIN {X 0,Y 420.859,Z 725.832,A -85,B 0,C 180,E1 -16506.35,E2 -16506.35} C_VEL
LIN {X 0,Y 424.008,Z 704.553,A -85,B 0,C 180,E1 -16507.645,E2 -16507.645} C_VEL
LIN {X 0,Y 426.552,Z 682.574,A -85,B 0,C 180,E1 -16508.7,E2 -16508.7} C_VEL
LIN {X 0,Y 428.685,Z 657.213,A -85,B 0,C 180,E1 -16509.616,E2 -16509.616} C_VEL
LIN {X 0,Y 432.655,Z 613.761,A -85,B 0,C 180,E1 -16510.882,E2 -16510.882} C_VEL
LIN {X 0,Y 438.249,Z 553.448,A -85,B 0,C 180,E1 -16512.359,E2 -16512.359} C_VEL
LIN {X 0,Y 442.721,Z 494.691,A -85,B 0,C 180,E1 -16513.592,E2 -16513.592} C_VEL
LIN {X 0,Y 446.474,Z 426.656,A -85,B 0,C 180,E1 -16514.778,E2 -16514.778} C_VEL
LIN {X 0,Y 447.694,Z 404.406,A -85,B 0,C 180,E1 -16515.163,E2 -16515.163} C_VEL
LIN {X 0,Y 453.87,Z 376.827,A -85,B 0,C 180,E1 -16516.178,E2 -16516.178} C_VEL
LIN {X 0,Y 454.278,Z 362.011,A -85,B 0,C 180,E1 -16517.232,E2 -16517.232} C_VEL
LIN {X 0,Y 447.684,Z 343.432,A -85,B 0,C 180,E1 -16519.805,E2 -16519.805} C_VEL
LIN {X 0,Y 440.52,Z 325.873,A -85,B 0,C 180,E1 -16522.533,E2 -16522.533} C_VEL
LIN {X 0,Y 434.093,Z 311.731,A -85,B 0,C 180,E1 -16525.002,E2 -16525.002} C_VEL
LIN {X 0,Y 426.278,Z 296.51,A -85,B 0,C 180,E1 -16527.987,E2 -16527.987} C_VEL
LIN {X 0,Y 419.921,Z 285.436,A -85,B 0,C 180,E1 -16530.469,E2 -16530.469} C_VEL
LIN {X 0,Y 414.738,Z 276.821,A -85,B 0,C 180,E1 -16532.582,E2 -16532.582} C_VEL
LIN {X 0,Y 411.157,Z 271.383,A -85,B 0,C 180,E1 -16534.079,E2 -16534.079} C_VEL
LIN {X 0,Y 407.9,Z 266.38,A -85,B 0,C 180,E1 -16535.526,E2 -16535.526} C_VEL
LIN {X 0,Y 405.036,Z 262.018,A -85,B 0,C 180,E1 -16536.85,E2 -16536.85} C_VEL
LIN {X 0,Y 401.5,Z 257.301,A -85,B 0,C 180,E1 -16538.525,E2 -16538.525} C_VEL
LIN {X 0,Y 400.444,Z 255.504,A -85,B 0,C 180,E1 -16539.08,E2 -16539.08} C_VEL
LIN {X 0,Y 397.56,Z 252.262,A -85,B 0,C 180,E1 -16540.496,E2 -16540.496} C_VEL
LIN {X 0,Y 396.257,Z 249.595,A -85,B 0,C 180,E1 -16541.309,E2 -16541.309} C_VEL
LIN {X 0,Y 393.207,Z 246.736,A -85,B 0,C 180,E1 -16542.92,E2 -16542.92} C_VEL
LIN {X 0,Y 391.725,Z 243.456,A -85,B 0,C 180,E1 -16543.998,E2 -16543.998} C_VEL
LIN {X 0,Y 388.66,Z 241.248,A -85,B 0,C 180,E1 -16545.777,E2 -16545.777} C_VEL
LIN {X 0,Y 387.021,Z 238.188,A -85,B 0,C 180,E1 -16547.125,E2 -16547.125} C_VEL
LIN {X 0,Y 386.776,Z 236.99,A -85,B 0,C 180,E1 -16547.534,E2 -16547.534} C_VEL
LIN {X 0,Y 386.785,Z 237.035,A -85,B 0,C 180,E1 -16551.526,E2 -16551.526} C_VEL
LIN {X 0,Y 386.777,Z 237.005,A -85,B 0,C 180,E1 -16555.552,E2 -16555.552} C_VEL
LIN {X 0,Y 386.783,Z 236.994,A -85,B 0,C 180,E1 -16559.556,E2 -16559.556} C_VEL
LIN {X 0,Y 386.784,Z 237.05,A -85,B 0,C 180,E1 -16563.557,E2 -16563.557} C_VEL
LIN {X 0,Y 386.786,Z 236.986,A -85,B 0,C 180,E1 -16567.576,E2 -16567.576} C_VEL
LIN {X 0,Y 386.785,Z 237.049,A -85,B 0,C 180,E1 -16571.633,E2 -16571.633} C_VEL
LIN {X 0,Y 386.804,Z 237.252,A -85,B 0,C 180,E1 -16572.997,E2 -16572.997} C_VEL
LIN {X 0,Y 388.187,Z 240.679,A -85,B 0,C 180,E1 -16573.86,E2 -16573.86} C_VEL
LIN {X 0,Y 389.427,Z 242.534,A -85,B 0,C 180,E1 -16574.422,E2 -16574.422} C_VEL
LIN {X 0,Y 391.397,Z 246.244,A -85,B 0,C 180,E1 -16575.408,E2 -16575.408} C_VEL
LIN {X 0,Y 395.007,Z 253.287,A -85,B 0,C 180,E1 -16577.227,E2 -16577.227} C_VEL
LIN {X 0,Y 399.489,Z 261.557,A -85,B 0,C 180,E1 -16579.292,E2 -16579.292} C_VEL
LIN {X 0,Y 406.761,Z 275.608,A -85,B 0,C 180,E1 -16582.549,E2 -16582.549} C_VEL
LIN {X 0,Y 414.763,Z 291.217,A -85,B 0,C 180,E1 -16585.871,E2 -16585.871} C_VEL
LIN {X 0,Y 424.484,Z 311.003,A -85,B 0,C 180,E1 -16589.648,E2 -16589.648} C_VEL
LIN {X 0,Y 433.421,Z 329.484,A -85,B 0,C 180,E1 -16592.79,E2 -16592.79} C_VEL
LIN {X 0,Y 452.32,Z 358.906,A -85,B 0,C 180,E1 -16595.801,E2 -16595.801} C_VEL
LIN {X 0,Y 455.523,Z 364.299,A -85,B 0,C 180,E1 -16596.29,E2 -16596.29} C_VEL
LIN {X 0,Y 438.872,Z 609.311,A -85,B 0,C 180,E1 -16601.176,E2 -16601.176} C_VEL
LIN {X 0,Y 433.695,Z 693.457,A -85,B 0,C 180,E1 -16602.902,E2 -16602.902} C_VEL
LIN {X 0,Y 431.196,Z 717.825,A -85,B 0,C 180,E1 -16603.614,E2 -16603.614} C_VEL
LIN {X 0,Y 427.945,Z 743.337,A -85,B 0,C 180,E1 -16604.598,E2 -16604.598} C_VEL
LIN {X 0,Y 424.437,Z 766.658,A -85,B 0,C 180,E1 -16605.739,E2 -16605.739} C_VEL
LIN {X 0,Y 420.604,Z 788.712,A -85,B 0,C 180,E1 -16607.071,E2 -16607.071} C_VEL
LIN {X 0,Y 416.379,Z 810.971,A -85,B 0,C 180,E1 -16608.671,E2 -16608.671} C_VEL
LIN {X 0,Y 412.115,Z 831.579,A -85,B 0,C 180,E1 -16610.44,E2 -16610.44} C_VEL
LIN {X 0,Y 407.434,Z 852.923,A -85,B 0,C 180,E1 -16612.599,E2 -16612.599} C_VEL
LIN {X 0,Y 403.261,Z 871.48,A -85,B 0,C 180,E1 -16614.796,E2 -16614.796} C_VEL
LIN {X 0,Y 399.203,Z 889.058,A -85,B 0,C 180,E1 -16617.247,E2 -16617.247} C_VEL
LIN {X 0,Y 395.414,Z 905.839,A -85,B 0,C 180,E1 -16619.955,E2 -16619.955} C_VEL
LIN {X 0,Y 392.287,Z 920.306,A -85,B 0,C 180,E1 -16622.691,E2 -16622.691} C_VEL
LIN {X 0,Y 389.531,Z 934.128,A -85,B 0,C 180,E1 -16625.751,E2 -16625.751} C_VEL
LIN {X 0,Y 387.573,Z 945.334,A -85,B 0,C 180,E1 -16628.669,E2 -16628.669} C_VEL
LIN {X 0,Y 386.099,Z 955.744,A -85,B 0,C 180,E1 -16631.895,E2 -16631.895} C_VEL
LIN {X 0,Y 385.254,Z 963.925,A -85,B 0,C 180,E1 -16634.957,E2 -16634.957} C_VEL
LIN {X 0,Y 384.815,Z 971.245,A -85,B 0,C 180,E1 -16638.404,E2 -16638.404} C_VEL
LIN {X 0,Y 384.768,Z 975.767,A -85,B 0,C 180,E1 -16641.181,E2 -16641.181} C_VEL
LIN {X 0,Y 384.887,Z 979.537,A -85,B 0,C 180,E1 -16644.335,E2 -16644.335} C_VEL
LIN {X 0,Y 385.007,Z 981.616,A -85,B 0,C 180,E1 -16647.47,E2 -16647.47} C_VEL
LIN {X 0,Y 385.054,Z 982.237,A -85,B 0,C 180,E1 -16650.149,E2 -16650.149} C_VEL
LIN {X 0,Y 384.962,Z 981.766,A -85,B 0,C 180,E1 -16652.829,E2 -16652.829} C_VEL
LIN {X 0,Y 384.793,Z 979.889,A -85,B 0,C 180,E1 -16655.966,E2 -16655.966} C_VEL
LIN {X 0,Y 384.661,Z 976.212,A -85,B 0,C 180,E1 -16659.275,E2 -16659.275} C_VEL
LIN {X 0,Y 384.754,Z 971.3,A -85,B 0,C 180,E1 -16662.457,E2 -16662.457} C_VEL
LIN {X 0,Y 385.317,Z 964.153,A -85,B 0,C 180,E1 -16665.966,E2 -16665.966} C_VEL
LIN {X 0,Y 386.425,Z 956.056,A -85,B 0,C 180,E1 -16669.186,E2 -16669.186} C_VEL
LIN {X 0,Y 388.557,Z 944.759,A -85,B 0,C 180,E1 -16672.889,E2 -16672.889} C_VEL
LIN {X 0,Y 391.457,Z 932.66,A -85,B 0,C 180,E1 -16676.225,E2 -16676.225} C_VEL
LIN {X 0,Y 395.148,Z 919.02,A -85,B 0,C 180,E1 -16679.4,E2 -16679.4} C_VEL
LIN {X 0,Y 399.86,Z 903.525,A -85,B 0,C 180,E1 -16682.523,E2 -16682.523} C_VEL
LIN {X 0,Y 405.323,Z 886.524,A -85,B 0,C 180,E1 -16685.431,E2 -16685.431} C_VEL
LIN {X 0,Y 411.794,Z 867.242,A -85,B 0,C 180,E1 -16688.256,E2 -16688.256} C_VEL
LIN {X 0,Y 418.532,Z 847.682,A -85,B 0,C 180,E1 -16690.708,E2 -16690.708} C_VEL
LIN {X 0,Y 425.937,Z 826.015,A -85,B 0,C 180,E1 -16692.996,E2 -16692.996} C_VEL
LIN {X 0,Y 433.473,Z 803.573,A -85,B 0,C 180,E1 -16694.992,E2 -16694.992} C_VEL
LIN {X 0,Y 441.288,Z 779.648,A -85,B 0,C 180,E1 -16696.758,E2 -16696.758} C_VEL
LIN {X 0,Y 448.406,Z 756.913,A -85,B 0,C 180,E1 -16698.14,E2 -16698.14} C_VEL
LIN {X 0,Y 455.78,Z 731.482,A -85,B 0,C 180,E1 -16699.381,E2 -16699.381} C_VEL
LIN {X 0,Y 462.797,Z 704.676,A -85,B 0,C 180,E1 -16700.375,E2 -16700.375} C_VEL
LIN {X 0,Y 469.158,Z 676.067,A -85,B 0,C 180,E1 -16701.166,E2 -16701.166} C_VEL
LIN {X 0,Y 476.133,Z 643.016,A -85,B 0,C 180,E1 -16701.995,E2 -16701.995} C_VEL
LIN {X 0,Y 462.977,Z 693.676,A -85,B 0,C 180,E1 -16703.593,E2 -16703.593} C_VEL
LIN {X 0,Y 456.058,Z 715.992,A -85,B 0,C 180,E1 -16704.479,E2 -16704.479} C_VEL
LIN {X 0,Y 448.511,Z 737.483,A -85,B 0,C 180,E1 -16705.588,E2 -16705.588} C_VEL
LIN {X 0,Y 440.185,Z 759.718,A -85,B 0,C 180,E1 -16707.041,E2 -16707.041} C_VEL
LIN {X 0,Y 431.751,Z 781.709,A -85,B 0,C 180,E1 -16708.828,E2 -16708.828} C_VEL
LIN {X 0,Y 423.949,Z 802.145,A -85,B 0,C 180,E1 -16710.854,E2 -16710.854} C_VEL
LIN {X 0,Y 417.034,Z 820.526,A -85,B 0,C 180,E1 -16713.054,E2 -16713.054} C_VEL
LIN {X 0,Y 410.915,Z 836.989,A -85,B 0,C 180,E1 -16715.411,E2 -16715.411} C_VEL
LIN {X 0,Y 405.68,Z 851.086,A -85,B 0,C 180,E1 -16717.846,E2 -16717.846} C_VEL
LIN {X 0,Y 401.228,Z 862.95,A -85,B 0,C 180,E1 -16720.34,E2 -16720.34} C_VEL
LIN {X 0,Y 397.481,Z 872.726,A -85,B 0,C 180,E1 -16722.883,E2 -16722.883} C_VEL
LIN {X 0,Y 394.521,Z 880.094,A -85,B 0,C 180,E1 -16725.319,E2 -16725.319} C_VEL
LIN {X 0,Y 392.095,Z 885.785,A -85,B 0,C 180,E1 -16727.78,E2 -16727.78} C_VEL
LIN {X 0,Y 389.965,Z 890.185,A -85,B 0,C 180,E1 -16730.555,E2 -16730.555} C_VEL
LIN {X 0,Y 388.387,Z 892.589,A -85,B 0,C 180,E1 -16733.347,E2 -16733.347} C_VEL
LIN {X 0,Y 387.318,Z 893.073,A -85,B 0,C 180,E1 -16736.003,E2 -16736.003} C_VEL
LIN {X 0,Y 386.62,Z 891.814,A -85,B 0,C 180,E1 -16738.666,E2 -16738.666} C_VEL
LIN {X 0,Y 386.227,Z 888.84,A -85,B 0,C 180,E1 -16741.335,E2 -16741.335} C_VEL
LIN {X 0,Y 386.098,Z 884.094,A -85,B 0,C 180,E1 -16744.01,E2 -16744.01} C_VEL
LIN {X 0,Y 386.253,Z 877.511,A -85,B 0,C 180,E1 -16746.69,E2 -16746.69} C_VEL
LIN {X 0,Y 386.708,Z 868.943,A -85,B 0,C 180,E1 -16749.375,E2 -16749.375} C_VEL
LIN {X 0,Y 387.48,Z 858.836,A -85,B 0,C 180,E1 -16751.914,E2 -16751.914} C_VEL
LIN {X 0,Y 388.564,Z 847.335,A -85,B 0,C 180,E1 -16754.302,E2 -16754.302} C_VEL
LIN {X 0,Y 390.022,Z 833.555,A -85,B 0,C 180,E1 -16756.686,E2 -16756.686} C_VEL
LIN {X 0,Y 391.77,Z 818.194,A -85,B 0,C 180,E1 -16758.913,E2 -16758.913} C_VEL
LIN {X 0,Y 393.77,Z 801.231,A -85,B 0,C 180,E1 -16760.98,E2 -16760.98} C_VEL
LIN {X 0,Y 395.966,Z 782.544,A -85,B 0,C 180,E1 -16762.885,E2 -16762.885} C_VEL
LIN {X 0,Y 398.192,Z 762.729,A -85,B 0,C 180,E1 -16764.556,E2 -16764.556} C_VEL
LIN {X 0,Y 400.469,Z 741.56,A -85,B 0,C 180,E1 -16766.017,E2 -16766.017} C_VEL
LIN {X 0,Y 402.655,Z 718.86,A -85,B 0,C 180,E1 -16767.268,E2 -16767.268} C_VEL
LIN {X 0,Y 404.637,Z 695.56,A -85,B 0,C 180,E1 -16768.253,E2 -16768.253} C_VEL
LIN {X 0,Y 406.317,Z 670.767,A -85,B 0,C 180,E1 -16768.999,E2 -16768.999} C_VEL
LIN {X 0,Y 416.368,Z 509.241,A -85,B 0,C 180,E1 -16773.05,E2 -16773.05} C_VEL
LIN {X 0,Y 411.819,Z 434.892,A -85,B 0,C 180,E1 -16775.728,E2 -16775.728} C_VEL
LIN {X 0,Y 417.311,Z 396.543,A -85,B 0,C 180,E1 -16779.076,E2 -16779.076} C_VEL
LIN {X 0,Y 419.025,Z 396.405,A -85,B 0,C 180,E1 -16779.401,E2 -16779.401} C_VEL
LIN {X 0,Y 422.554,Z 393.983,A -85,B 0,C 180,E1 -16779.887,E2 -16779.887} C_VEL
LIN {X 0,Y 426.507,Z 390.073,A -85,B 0,C 180,E1 -16780.32,E2 -16780.32} C_VEL
LIN {X 0,Y 429.92,Z 388.343,A -85,B 0,C 180,E1 -16780.809,E2 -16780.809} C_VEL
LIN {X 0,Y 434.535,Z 384.439,A -85,B 0,C 180,E1 -16781.331,E2 -16781.331} C_VEL
LIN {X 0,Y 436.012,Z 383.401,A -85,B 0,C 180,E1 -16781.51,E2 -16781.51} C_VEL
LIN {X 0,Y 441.133,Z 380.207,A -85,B 0,C 180,E1 -16782.139,E2 -16782.139} C_VEL
LIN {X 0,Y 444.314,Z 377.511,A -85,B 0,C 180,E1 -16782.464,E2 -16782.464} C_VEL
LIN {X 0,Y 450.224,Z 373.917,A -85,B 0,C 180,E1 -16783.16,E2 -16783.16} C_VEL
LIN {X 0,Y 453.541,Z 371.552,A -85,B 0,C 180,E1 -16783.504,E2 -16783.504} C_VEL
LIN {X 0,Y 453.879,Z 371.446,A -85,B 0,C 180,E1 -16783.549,E2 -16783.549} C_VEL
LIN {X 0,Y 453.587,Z 377.698,A -85,B 0,C 180,E1 -16783.967,E2 -16783.967} C_VEL
LIN {X 0,Y 447.352,Z 406.224,A -85,B 0,C 180,E1 -16784.989,E2 -16784.989} C_VEL
LIN {X 0,Y 443.108,Z 487.162,A -85,B 0,C 180,E1 -16786.367,E2 -16786.367} C_VEL
LIN {X 0,Y 438.689,Z 547.175,A -85,B 0,C 180,E1 -16787.603,E2 -16787.603} C_VEL
LIN {X 0,Y 433.081,Z 608.665,A -85,B 0,C 180,E1 -16789.088,E2 -16789.088} C_VEL
LIN {X 0,Y 428.889,Z 653.731,A -85,B 0,C 180,E1 -16790.374,E2 -16790.374} C_VEL
LIN {X 0,Y 426.647,Z 680.87,A -85,B 0,C 180,E1 -16791.333,E2 -16791.333} C_VEL
LIN {X 0,Y 424.281,Z 701.902,A -85,B 0,C 180,E1 -16792.317,E2 -16792.317} C_VEL
LIN {X 0,Y 421.328,Z 722.527,A -85,B 0,C 180,E1 -16793.532,E2 -16793.532} C_VEL
LIN {X 0,Y 417.968,Z 742.211,A -85,B 0,C 180,E1 -16794.96,E2 -16794.96} C_VEL
LIN {X 0,Y 414.191,Z 761.378,A -85,B 0,C 180,E1 -16796.645,E2 -16796.645} C_VEL
LIN {X 0,Y 410.178,Z 779.564,A -85,B 0,C 180,E1 -16798.561,E2 -16798.561} C_VEL
LIN {X 0,Y 406.046,Z 796.826,A -85,B 0,C 180,E1 -16800.738,E2 -16800.738} C_VEL
LIN {X 0,Y 402.086,Z 812.466,A -85,B 0,C 180,E1 -16803.09,E2 -16803.09} C_VEL
LIN {X 0,Y 398.304,Z 826.924,A -85,B 0,C 180,E1 -16805.688,E2 -16805.688} C_VEL
LIN {X 0,Y 394.918,Z 839.765,A -85,B 0,C 180,E1 -16808.462,E2 -16808.462} C_VEL
LIN {X 0,Y 392.014,Z 851.002,A -85,B 0,C 180,E1 -16811.408,E2 -16811.408} C_VEL
LIN {X 0,Y 391.69,Z 852.277,A -85,B 0,C 180,E1 -16811.788,E2 -16811.788} C_VEL
LIN {X 0,Y 389.915,Z 855.755,A -85,B 0,C 180,E1 -16812.777,E2 -16812.777} C_VEL
LIN {X 0,Y 381.987,Z 864.585,A -85,B 0,C 180,E1 -16815.391,E2 -16815.391} C_VEL
LIN {X 0,Y 380.731,Z 866.883,A -85,B 0,C 180,E1 -16816.312,E2 -16816.312} C_VEL
LIN {X 0,Y 379.318,Z 873.312,A -85,B 0,C 180,E1 -16819.52,E2 -16819.52} C_VEL
LIN {X 0,Y 378.415,Z 878.087,A -85,B 0,C 180,E1 -16822.866,E2 -16822.866} C_VEL
LIN {X 0,Y 377.961,Z 880.797,A -85,B 0,C 180,E1 -16825.904,E2 -16825.904} C_VEL
LIN {X 0,Y 377.77,Z 882.092,A -85,B 0,C 180,E1 -16829.09,E2 -16829.09} C_VEL
LIN {X 0,Y 377.819,Z 881.851,A -85,B 0,C 180,E1 -16832.123,E2 -16832.123} C_VEL
LIN {X 0,Y 378.106,Z 880.012,A -85,B 0,C 180,E1 -16835.311,E2 -16835.311} C_VEL
LIN {X 0,Y 378.69,Z 876.473,A -85,B 0,C 180,E1 -16838.503,E2 -16838.503} C_VEL
LIN {X 0,Y 379.696,Z 871.459,A -85,B 0,C 180,E1 -16841.585,E2 -16841.585} C_VEL
LIN {X 0,Y 381.253,Z 864.611,A -85,B 0,C 180,E1 -16844.738,E2 -16844.738} C_VEL
LIN {X 0,Y 383.432,Z 855.952,A -85,B 0,C 180,E1 -16847.856,E2 -16847.856} C_VEL
LIN {X 0,Y 386.143,Z 845.81,A -85,B 0,C 180,E1 -16850.806,E2 -16850.806} C_VEL
LIN {X 0,Y 389.371,Z 834.087,A -85,B 0,C 180,E1 -16853.616,E2 -16853.616} C_VEL
LIN {X 0,Y 393.059,Z 820.771,A -85,B 0,C 180,E1 -16856.272,E2 -16856.272} C_VEL
LIN {X 0,Y 397.211,Z 805.365,A -85,B 0,C 180,E1 -16858.834,E2 -16858.834} C_VEL
LIN {X 0,Y 401.443,Z 788.927,A -85,B 0,C 180,E1 -16861.12,E2 -16861.12} C_VEL
LIN {X 0,Y 405.661,Z 771.278,A -85,B 0,C 180,E1 -16863.175,E2 -16863.175} C_VEL
LIN {X 0,Y 409.732,Z 752.541,A -85,B 0,C 180,E1 -16864.993,E2 -16864.993} C_VEL
LIN {X 0,Y 413.555,Z 732.404,A -85,B 0,C 180,E1 -16866.61,E2 -16866.61} C_VEL
LIN {X 0,Y 416.899,Z 711.64,A -85,B 0,C 180,E1 -16867.966,E2 -16867.966} C_VEL
LIN {X 0,Y 419.68,Z 689.938,A -85,B 0,C 180,E1 -16869.096,E2 -16869.096} C_VEL
LIN {X 0,Y 421.825,Z 667.382,A -85,B 0,C 180,E1 -16869.991,E2 -16869.991} C_VEL
LIN {X 0,Y 425.72,Z 623.989,A -85,B 0,C 180,E1 -16871.327,E2 -16871.327} C_VEL
LIN {X 0,Y 431.631,Z 563.511,A -85,B 0,C 180,E1 -16872.864,E2 -16872.864} C_VEL
LIN {X 0,Y 436.608,Z 501.534,A -85,B 0,C 180,E1 -16874.199,E2 -16874.199} C_VEL
LIN {X 0,Y 440.103,Z 442.423,A -85,B 0,C 180,E1 -16875.26,E2 -16875.26} C_VEL
LIN {X 0,Y 442.011,Z 407.151,A -85,B 0,C 180,E1 -16875.862,E2 -16875.862} C_VEL
LIN {X 0,Y 448.465,Z 378.513,A -85,B 0,C 180,E1 -16876.912,E2 -16876.912} C_VEL
LIN {X 0,Y 448.812,Z 366.097,A -85,B 0,C 180,E1 -16877.801,E2 -16877.801} C_VEL
LIN {X 0,Y 442.169,Z 347.278,A -85,B 0,C 180,E1 -16880.454,E2 -16880.454} C_VEL
LIN {X 0,Y 435.242,Z 330.249,A -85,B 0,C 180,E1 -16883.158,E2 -16883.158} C_VEL
LIN {X 0,Y 429.223,Z 316.975,A -85,B 0,C 180,E1 -16885.523,E2 -16885.523} C_VEL
LIN {X 0,Y 423.212,Z 305.007,A -85,B 0,C 180,E1 -16887.887,E2 -16887.887} C_VEL
LIN {X 0,Y 416.718,Z 293.035,A -85,B 0,C 180,E1 -16890.535,E2 -16890.535} C_VEL
LIN {X 0,Y 410.973,Z 283.436,A -85,B 0,C 180,E1 -16892.937,E2 -16892.937} C_VEL
LIN {X 0,Y 407.293,Z 277.723,A -85,B 0,C 180,E1 -16894.556,E2 -16894.556} C_VEL
LIN {X 0,Y 404.436,Z 273.266,A -85,B 0,C 180,E1 -16895.847,E2 -16895.847} C_VEL
LIN {X 0,Y 400.989,Z 268.067,A -85,B 0,C 180,E1 -16897.495,E2 -16897.495} C_VEL
LIN {X 0,Y 398.189,Z 264.051,A -85,B 0,C 180,E1 -16898.917,E2 -16898.917} C_VEL
LIN {X 0,Y 397.363,Z 262.698,A -85,B 0,C 180,E1 -16899.373,E2 -16899.373} C_VEL
LIN {X 0,Y 394.418,Z 259.15,A -85,B 0,C 180,E1 -16900.873,E2 -16900.873} C_VEL
LIN {X 0,Y 393.235,Z 256.865,A -85,B 0,C 180,E1 -16901.621,E2 -16901.621} C_VEL
LIN {X 0,Y 390.311,Z 253.852,A -85,B 0,C 180,E1 -16903.25,E2 -16903.25} C_VEL
LIN {X 0,Y 388.842,Z 250.863,A -85,B 0,C 180,E1 -16904.335,E2 -16904.335} C_VEL
LIN {X 0,Y 385.83,Z 248.32,A -85,B 0,C 180,E1 -16906.207,E2 -16906.207} C_VEL
LIN {X 0,Y 384.268,Z 244.981,A -85,B 0,C 180,E1 -16907.604,E2 -16907.604} C_VEL
LIN {X 0,Y 383.812,Z 244.424,A -85,B 0,C 180,E1 -16907.971,E2 -16907.971} C_VEL
LIN {X 0,Y 380.385,Z 241.855,A -85,B 0,C 180,E1 -16910.773,E2 -16910.773} C_VEL
LIN {X 0,Y 378.93,Z 238.588,A -85,B 0,C 180,E1 -16912.647,E2 -16912.647} C_VEL
LIN {X 0,Y 378.849,Z 237.983,A -85,B 0,C 180,E1 -16913.027,E2 -16913.027} C_VEL
LIN {X 0,Y 378.843,Z 238.041,A -85,B 0,C 180,E1 -16917.126,E2 -16917.126} C_VEL
LIN {X 0,Y 378.842,Z 237.977,A -85,B 0,C 180,E1 -16921.21,E2 -16921.21} C_VEL
LIN {X 0,Y 378.842,Z 237.999,A -85,B 0,C 180,E1 -16925.3,E2 -16925.3} C_VEL
LIN {X 0,Y 378.842,Z 238.004,A -85,B 0,C 180,E1 -16929.265,E2 -16929.265} C_VEL
LIN {X 0,Y 378.872,Z 238.232,A -85,B 0,C 180,E1 -16931.339,E2 -16931.339} C_VEL
LIN {X 0,Y 380.071,Z 241.43,A -85,B 0,C 180,E1 -16932.15,E2 -16932.15} C_VEL
LIN {X 0,Y 381.612,Z 243.662,A -85,B 0,C 180,E1 -16932.869,E2 -16932.869} C_VEL
LIN {X 0,Y 383.464,Z 247.268,A -85,B 0,C 180,E1 -16933.88,E2 -16933.88} C_VEL
LIN {X 0,Y 387.079,Z 254.192,A -85,B 0,C 180,E1 -16935.738,E2 -16935.738} C_VEL
LIN {X 0,Y 389.937,Z 259.625,A -85,B 0,C 180,E1 -16937.151,E2 -16937.151} C_VEL
LIN {X 0,Y 394.087,Z 267.357,A -85,B 0,C 180,E1 -16939.105,E2 -16939.105} C_VEL
LIN {X 0,Y 401.388,Z 281.511,A -85,B 0,C 180,E1 -16942.404,E2 -16942.404} C_VEL
LIN {X 0,Y 409.092,Z 296.602,A -85,B 0,C 180,E1 -16945.634,E2 -16945.634} C_VEL
LIN {X 0,Y 418.828,Z 316.5,A -85,B 0,C 180,E1 -16949.459,E2 -16949.459} C_VEL
LIN {X 0,Y 425.734,Z 330.733,A -85,B 0,C 180,E1 -16951.9,E2 -16951.9} C_VEL
LIN {X 0,Y 445.624,Z 361.563,A -85,B 0,C 180,E1 -16955.137,E2 -16955.137} C_VEL
LIN {X 0,Y 449.153,Z 367.707,A -85,B 0,C 180,E1 -16955.703,E2 -16955.703} C_VEL
LIN {X 0,Y 431.295,Z 623.048,A -85,B 0,C 180,E1 -16960.884,E2 -16960.884} C_VEL
LIN {X 0,Y 426.757,Z 693.714,A -85,B 0,C 180,E1 -16962.373,E2 -16962.373} C_VEL
LIN {X 0,Y 424.171,Z 718.167,A -85,B 0,C 180,E1 -16963.102,E2 -16963.102} C_VEL
LIN {X 0,Y 420.933,Z 742.907,A -85,B 0,C 180,E1 -16964.074,E2 -16964.074} C_VEL
LIN {X 0,Y 417.501,Z 765.209,A -85,B 0,C 180,E1 -16965.175,E2 -16965.175} C_VEL
LIN {X 0,Y 413.448,Z 788.171,A -85,B 0,C 180,E1 -16966.571,E2 -16966.571} C_VEL
LIN {X 0,Y 409.206,Z 810.052,A -85,B 0,C 180,E1 -16968.159,E2 -16968.159} C_VEL
LIN {X 0,Y 404.799,Z 830.866,A -85,B 0,C 180,E1 -16969.972,E2 -16969.972} C_VEL
LIN {X 0,Y 399.952,Z 852.42,A -85,B 0,C 180,E1 -16972.187,E2 -16972.187} C_VEL
LIN {X 0,Y 395.562,Z 871.48,A -85,B 0,C 180,E1 -16974.483,E2 -16974.483} C_VEL
LIN {X 0,Y 391.342,Z 889.34,A -85,B 0,C 180,E1 -16977.029,E2 -16977.029} C_VEL
LIN {X 0,Y 387.295,Z 906.832,A -85,B 0,C 180,E1 -16979.944,E2 -16979.944} C_VEL
LIN {X 0,Y 384.312,Z 920.375,A -85,B 0,C 180,E1 -16982.58,E2 -16982.58} C_VEL
LIN {X 0,Y 381.524,Z 934.074,A -85,B 0,C 180,E1 -16985.703,E2 -16985.703} C_VEL
LIN {X 0,Y 379.464,Z 945.788,A -85,B 0,C 180,E1 -16988.839,E2 -16988.839} C_VEL
LIN {X 0,Y 378.08,Z 955.501,A -85,B 0,C 180,E1 -16991.976,E2 -16991.976} C_VEL
LIN {X 0,Y 377.253,Z 963.595,A -85,B 0,C 180,E1 -16995.102,E2 -16995.102} C_VEL
LIN {X 0,Y 376.854,Z 970.579,A -85,B 0,C 180,E1 -16998.522,E2 -16998.522} C_VEL
LIN {X 0,Y 376.824,Z 974.966,A -85,B 0,C 180,E1 -17001.301,E2 -17001.301} C_VEL
LIN {X 0,Y 376.955,Z 978.678,A -85,B 0,C 180,E1 -17004.52,E2 -17004.52} C_VEL
LIN {X 0,Y 377.088,Z 980.675,A -85,B 0,C 180,E1 -17007.721,E2 -17007.721} C_VEL
LIN {X 0,Y 377.105,Z 981.226,A -85,B 0,C 180,E1 -17010.456,E2 -17010.456} C_VEL
LIN {X 0,Y 377.003,Z 980.629,A -85,B 0,C 180,E1 -17013.345,E2 -17013.345} C_VEL
LIN {X 0,Y 376.787,Z 978.379,A -85,B 0,C 180,E1 -17016.705,E2 -17016.705} C_VEL
LIN {X 0,Y 376.681,Z 974.912,A -85,B 0,C 180,E1 -17019.781,E2 -17019.781} C_VEL
LIN {X 0,Y 376.839,Z 969.657,A -85,B 0,C 180,E1 -17023.191,E2 -17023.191} C_VEL
LIN {X 0,Y 377.529,Z 962.292,A -85,B 0,C 180,E1 -17026.78,E2 -17026.78} C_VEL
LIN {X 0,Y 378.89,Z 953.664,A -85,B 0,C 180,E1 -17030.225,E2 -17030.225} C_VEL
LIN {X 0,Y 381.225,Z 942.664,A -85,B 0,C 180,E1 -17033.823,E2 -17033.823} C_VEL
LIN {X 0,Y 384.464,Z 930.371,A -85,B 0,C 180,E1 -17037.241,E2 -17037.241} C_VEL
LIN {X 0,Y 388.547,Z 916.635,A -85,B 0,C 180,E1 -17040.462,E2 -17040.462} C_VEL
LIN {X 0,Y 393.954,Z 900.197,A -85,B 0,C 180,E1 -17043.769,E2 -17043.769} C_VEL
LIN {X 0,Y 399.68,Z 883.887,A -85,B 0,C 180,E1 -17046.577,E2 -17046.577} C_VEL
LIN {X 0,Y 406.563,Z 864.805,A -85,B 0,C 180,E1 -17049.384,E2 -17049.384} C_VEL
LIN {X 0,Y 414.428,Z 843.55,A -85,B 0,C 180,E1 -17052.03,E2 -17052.03} C_VEL
LIN {X 0,Y 422.162,Z 822.68,A -85,B 0,C 180,E1 -17054.229,E2 -17054.229} C_VEL
LIN {X 0,Y 430.479,Z 799.67,A -85,B 0,C 180,E1 -17056.251,E2 -17056.251} C_VEL
LIN {X 0,Y 439.113,Z 775.1,A -85,B 0,C 180,E1 -17058.027,E2 -17058.027} C_VEL
LIN {X 0,Y 447.335,Z 750.521,A -85,B 0,C 180,E1 -17059.462,E2 -17059.462} C_VEL
LIN {X 0,Y 454.928,Z 726.213,A -85,B 0,C 180,E1 -17060.585,E2 -17060.585} C_VEL
LIN {X 0,Y 462.045,Z 701.015,A -85,B 0,C 180,E1 -17061.472,E2 -17061.472} C_VEL
LIN {X 0,Y 467.431,Z 678.924,A -85,B 0,C 180,E1 -17062.092,E2 -17062.092} C_VEL
LIN {X 0,Y 460.127,Z 703.41,A -85,B 0,C 180,E1 -17062.913,E2 -17062.913} C_VEL
LIN {X 0,Y 452.805,Z 723.987,A -85,B 0,C 180,E1 -17063.793,E2 -17063.793} C_VEL
LIN {X 0,Y 444.322,Z 745.531,A -85,B 0,C 180,E1 -17064.981,E2 -17064.981} C_VEL
LIN {X 0,Y 435.095,Z 767.549,A -85,B 0,C 180,E1 -17066.527,E2 -17066.527} C_VEL
LIN {X 0,Y 425.825,Z 789.229,A -85,B 0,C 180,E1 -17068.424,E2 -17068.424} C_VEL
LIN {X 0,Y 417.313,Z 809.369,A -85,B 0,C 180,E1 -17070.581,E2 -17070.581} C_VEL
LIN {X 0,Y 409.631,Z 828.003,A -85,B 0,C 180,E1 -17072.998,E2 -17072.998} C_VEL
LIN {X 0,Y 403.38,Z 843.309,A -85,B 0,C 180,E1 -17075.39,E2 -17075.39} C_VEL
LIN {X 0,Y 397.742,Z 857.099,A -85,B 0,C 180,E1 -17078.002,E2 -17078.002} C_VEL
LIN {X 0,Y 393.218,Z 868.031,A -85,B 0,C 180,E1 -17080.542,E2 -17080.542} C_VEL
LIN {X 0,Y 389.213,Z 877.396,A -85,B 0,C 180,E1 -17083.278,E2 -17083.278} C_VEL
LIN {X 0,Y 386.092,Z 884.31,A -85,B 0,C 180,E1 -17085.91,E2 -17085.91} C_VEL
LIN {X 0,Y 383.585,Z 889.38,A -85,B 0,C 180,E1 -17088.574,E2 -17088.574} C_VEL
LIN {X 0,Y 381.549,Z 892.794,A -85,B 0,C 180,E1 -17091.409,E2 -17091.409} C_VEL
LIN {X 0,Y 380.19,Z 894.18,A -85,B 0,C 180,E1 -17093.961,E2 -17093.961} C_VEL
LIN {X 0,Y 379.178,Z 894.027,A -85,B 0,C 180,E1 -17096.674,E2 -17096.674} C_VEL
LIN {X 0,Y 378.542,Z 892.117,A -85,B 0,C 180,E1 -17099.395,E2 -17099.395} C_VEL
LIN {X 0,Y 378.201,Z 888.493,A -85,B 0,C 180,E1 -17102.121,E2 -17102.121} C_VEL
LIN {X 0,Y 378.151,Z 883.073,A -85,B 0,C 180,E1 -17104.854,E2 -17104.854} C_VEL
LIN {X 0,Y 378.383,Z 876.257,A -85,B 0,C 180,E1 -17107.44,E2 -17107.44} C_VEL
LIN {X 0,Y 378.947,Z 866.932,A -85,B 0,C 180,E1 -17110.198,E2 -17110.198} C_VEL
LIN {X 0,Y 379.849,Z 856.175,A -85,B 0,C 180,E1 -17112.775,E2 -17112.775} C_VEL
LIN {X 0,Y 381.079,Z 843.917,A -85,B 0,C 180,E1 -17115.212,E2 -17115.212} C_VEL
LIN {X 0,Y 382.655,Z 829.783,A -85,B 0,C 180,E1 -17117.566,E2 -17117.566} C_VEL
LIN {X 0,Y 384.504,Z 814.134,A -85,B 0,C 180,E1 -17119.759,E2 -17119.759} C_VEL
LIN {X 0,Y 386.67,Z 796.201,A -85,B 0,C 180,E1 -17121.862,E2 -17121.862} C_VEL
LIN {X 0,Y 388.93,Z 777.179,A -85,B 0,C 180,E1 -17123.725,E2 -17123.725} C_VEL
LIN {X 0,Y 391.231,Z 757.207,A -85,B 0,C 180,E1 -17125.346,E2 -17125.346} C_VEL
LIN {X 0,Y 393.485,Z 736.399,A -85,B 0,C 180,E1 -17126.73,E2 -17126.73} C_VEL
LIN {X 0,Y 395.641,Z 713.888,A -85,B 0,C 180,E1 -17127.916,E2 -17127.916} C_VEL
LIN {X 0,Y 397.561,Z 690.842,A -85,B 0,C 180,E1 -17128.839,E2 -17128.839} C_VEL
LIN {X 0,Y 399.673,Z 658.334,A -85,B 0,C 180,E1 -17129.764,E2 -17129.764} C_VEL
LIN {X 0,Y 409.338,Z 509.955,A -85,B 0,C 180,E1 -17133.579,E2 -17133.579} C_VEL
LIN {X 0,Y 404.878,Z 434.229,A -85,B 0,C 180,E1 -17136.349,E2 -17136.349} C_VEL
LIN {X 0,Y 408.253,Z 410.899,A -85,B 0,C 180,E1 -17138.414,E2 -17138.414} C_VEL
LIN {X 0,Y 410.174,Z 410.673,A -85,B 0,C 180,E1 -17138.792,E2 -17138.792} C_VEL
LIN {X 0,Y 413.693,Z 408.067,A -85,B 0,C 180,E1 -17139.291,E2 -17139.291} C_VEL
LIN {X 0,Y 417.643,Z 403.908,A -85,B 0,C 180,E1 -17139.735,E2 -17139.735} C_VEL
LIN {X 0,Y 420.991,Z 402.172,A -85,B 0,C 180,E1 -17140.243,E2 -17140.243} C_VEL
LIN {X 0,Y 425.545,Z 398.227,A -85,B 0,C 180,E1 -17140.784,E2 -17140.784} C_VEL
LIN {X 0,Y 427.093,Z 396.825,A -85,B 0,C 180,E1 -17140.96,E2 -17140.96} C_VEL
LIN {X 0,Y 432.087,Z 393.697,A -85,B 0,C 180,E1 -17141.617,E2 -17141.617} C_VEL
LIN {X 0,Y 436.002,Z 390.332,A -85,B 0,C 180,E1 -17142.04,E2 -17142.04} C_VEL
LIN {X 0,Y 441.889,Z 386.617,A -85,B 0,C 180,E1 -17142.753,E2 -17142.753} C_VEL
LIN {X 0,Y 445.028,Z 384.06,A -85,B 0,C 180,E1 -17143.081,E2 -17143.081} C_VEL
LIN {X 0,Y 447.297,Z 382.973,A -85,B 0,C 180,E1 -17143.368,E2 -17143.368} C_VEL
LIN {X 0,Y 441.667,Z 409.03,A -85,B 0,C 180,E1 -17144.29,E2 -17144.29} C_VEL
LIN {X 0,Y 437.314,Z 489.547,A -85,B 0,C 180,E1 -17145.671,E2 -17145.671} C_VEL
LIN {X 0,Y 432.777,Z 549.361,A -85,B 0,C 180,E1 -17146.915,E2 -17146.915} C_VEL
LIN {X 0,Y 426.969,Z 611.022,A -85,B 0,C 180,E1 -17148.423,E2 -17148.423} C_VEL
LIN {X 0,Y 422.69,Z 655.453,A -85,B 0,C 180,E1 -17149.719,E2 -17149.719} C_VEL
LIN {X 0,Y 420.372,Z 682.454,A -85,B 0,C 180,E1 -17150.689,E2 -17150.689} C_VEL
LIN {X 0,Y 418.051,Z 702.567,A -85,B 0,C 180,E1 -17151.638,E2 -17151.638} C_VEL
LIN {X 0,Y 414.965,Z 723.485,A -85,B 0,C 180,E1 -17152.88,E2 -17152.88} C_VEL
LIN {X 0,Y 411.486,Z 743.206,A -85,B 0,C 180,E1 -17154.325,E2 -17154.325} C_VEL
LIN {X 0,Y 407.506,Z 762.686,A -85,B 0,C 180,E1 -17156.059,E2 -17156.059} C_VEL
LIN {X 0,Y 403.42,Z 780.555,A -85,B 0,C 180,E1 -17157.967,E2 -17157.967} C_VEL
LIN {X 0,Y 399.115,Z 797.862,A -85,B 0,C 180,E1 -17160.179,E2 -17160.179} C_VEL
LIN {X 0,Y 394.99,Z 813.492,A -85,B 0,C 180,E1 -17162.566,E2 -17162.566} C_VEL
LIN {X 0,Y 391.041,Z 827.948,A -85,B 0,C 180,E1 -17165.206,E2 -17165.206} C_VEL
LIN {X 0,Y 387.496,Z 840.784,A -85,B 0,C 180,E1 -17168.028,E2 -17168.028} C_VEL
LIN {X 0,Y 384.448,Z 852.02,A -85,B 0,C 180,E1 -17171.028,E2 -17171.028} C_VEL
LIN {X 0,Y 382.074,Z 861.207,A -85,B 0,C 180,E1 -17174.051,E2 -17174.051} C_VEL
LIN {X 0,Y 380.731,Z 866.883,A -85,B 0,C 180,E1 -17176.312,E2 -17176.312} C_VEL
LIN {X 0,Y 379.21,Z 869.447,A -85,B 0,C 180,E1 -17177.396,E2 -17177.396} C_VEL
LIN {X 0,Y 371.898,Z 875.806,A -85,B 0,C 180,E1 -17180.283,E2 -17180.283} C_VEL
LIN {X 0,Y 370.852,Z 877.297,A -85,B 0,C 180,E1 -17181.273,E2 -17181.273} C_VEL
LIN {X 0,Y 370.201,Z 880.928,A -85,B 0,C 180,E1 -17184.575,E2 -17184.575} C_VEL
LIN {X 0,Y 369.888,Z 882.807,A -85,B 0,C 180,E1 -17187.831,E2 -17187.831} C_VEL
LIN {X 0,Y 369.83,Z 883.108,A -85,B 0,C 180,E1 -17190.929,E2 -17190.929} C_VEL
LIN {X 0,Y 370.03,Z 881.872,A -85,B 0,C 180,E1 -17194.184,E2 -17194.184} C_VEL
LIN {X 0,Y 370.54,Z 879.03,A -85,B 0,C 180,E1 -17197.442,E2 -17197.442} C_VEL
LIN {X 0,Y 371.46,Z 874.454,A -85,B 0,C 180,E1 -17200.733,E2 -17200.733} C_VEL
LIN {X 0,Y 372.927,Z 868.165,A -85,B 0,C 180,E1 -17203.964,E2 -17203.964} C_VEL
LIN {X 0,Y 374.905,Z 860.388,A -85,B 0,C 180,E1 -17207.06,E2 -17207.06} C_VEL
LIN {X 0,Y 377.56,Z 850.76,A -85,B 0,C 180,E1 -17210.138,E2 -17210.138} C_VEL
LIN {X 0,Y 380.727,Z 839.683,A -85,B 0,C 180,E1 -17213.036,E2 -17213.036} C_VEL
LIN {X 0,Y 384.34,Z 827.194,A -85,B 0,C 180,E1 -17215.751,E2 -17215.751} C_VEL
LIN {X 0,Y 388.302,Z 813.313,A -85,B 0,C 180,E1 -17218.282,E2 -17218.282} C_VEL
LIN {X 0,Y 392.51,Z 798.005,A -85,B 0,C 180,E1 -17220.629,E2 -17220.629} C_VEL
LIN {X 0,Y 396.862,Z 781.154,A -85,B 0,C 180,E1 -17222.799,E2 -17222.799} C_VEL
LIN {X 0,Y 401.131,Z 763.186,A -85,B 0,C 180,E1 -17224.735,E2 -17224.735} C_VEL
LIN {X 0,Y 405.254,Z 743.612,A -85,B 0,C 180,E1 -17226.486,E2 -17226.486} C_VEL
LIN {X 0,Y 408.889,Z 723.656,A -85,B 0,C 180,E1 -17227.953,E2 -17227.953} C_VEL
LIN {X 0,Y 412.071,Z 702.557,A -85,B 0,C 180,E1 -17229.205,E2 -17229.205} C_VEL
LIN {X 0,Y 414.643,Z 680.459,A -85,B 0,C 180,E1 -17230.232,E2 -17230.232} C_VEL
LIN {X 0,Y 417.74,Z 645.31,A -85,B 0,C 180,E1 -17231.439,E2 -17231.439} C_VEL
LIN {X 0,Y 423.364,Z 590.497,A -85,B 0,C 180,E1 -17232.961,E2 -17232.961} C_VEL
LIN {X 0,Y 428.981,Z 528.55,A -85,B 0,C 180,E1 -17234.402,E2 -17234.402} C_VEL
LIN {X 0,Y 432.839,Z 473.766,A -85,B 0,C 180,E1 -17235.481,E2 -17235.481} C_VEL
LIN {X 0,Y 436.393,Z 409.894,A -85,B 0,C 180,E1 -17236.579,E2 -17236.579} C_VEL
LIN {X 0,Y 443.125,Z 379.736,A -85,B 0,C 180,E1 -17237.693,E2 -17237.693} C_VEL
LIN {X 0,Y 443.418,Z 370.191,A -85,B 0,C 180,E1 -17238.387,E2 -17238.387} C_VEL
LIN {X 0,Y 436.975,Z 351.876,A -85,B 0,C 180,E1 -17241.004,E2 -17241.004} C_VEL
LIN {X 0,Y 430.35,Z 335.39,A -85,B 0,C 180,E1 -17243.667,E2 -17243.667} C_VEL
LIN {X 0,Y 423.53,Z 320.133,A -85,B 0,C 180,E1 -17246.465,E2 -17246.465} C_VEL
LIN {X 0,Y 416.8,Z 306.982,A -85,B 0,C 180,E1 -17249.186,E2 -17249.186} C_VEL
LIN {X 0,Y 410.43,Z 295.258,A -85,B 0,C 180,E1 -17251.953,E2 -17251.953} C_VEL
LIN {X 0,Y 404.335,Z 285.234,A -85,B 0,C 180,E1 -17254.671,E2 -17254.671} C_VEL
LIN {X 0,Y 400.776,Z 279.844,A -85,B 0,C 180,E1 -17256.294,E2 -17256.294} C_VEL
LIN {X 0,Y 397.678,Z 275.026,A -85,B 0,C 180,E1 -17257.843,E2 -17257.843} C_VEL
LIN {X 0,Y 394.835,Z 270.674,A -85,B 0,C 180,E1 -17259.351,E2 -17259.351} C_VEL
LIN {X 0,Y 391.2,Z 265.823,A -85,B 0,C 180,E1 -17261.329,E2 -17261.329} C_VEL
LIN {X 0,Y 390.26,Z 264.119,A -85,B 0,C 180,E1 -17261.94,E2 -17261.94} C_VEL
LIN {X 0,Y 387.368,Z 260.8,A -85,B 0,C 180,E1 -17263.659,E2 -17263.659} C_VEL
LIN {X 0,Y 386.217,Z 258.366,A -85,B 0,C 180,E1 -17264.534,E2 -17264.534} C_VEL
LIN {X 0,Y 383.219,Z 255.642,A -85,B 0,C 180,E1 -17266.495,E2 -17266.495} C_VEL
LIN {X 0,Y 381.584,Z 252.095,A -85,B 0,C 180,E1 -17268.053,E2 -17268.053} C_VEL
LIN {X 0,Y 378.174,Z 249.532,A -85,B 0,C 180,E1 -17270.872,E2 -17270.872} C_VEL
LIN {X 0,Y 376.726,Z 246.121,A -85,B 0,C 180,E1 -17272.911,E2 -17272.911} C_VEL
LIN {X 0,Y 376.458,Z 245.616,A -85,B 0,C 180,E1 -17273.289,E2 -17273.289} C_VEL
LIN {X 0,Y 372.699,Z 243.102,A -85,B 0,C 180,E1 -17281.23,E2 -17281.23} C_VEL
LIN {X 0,Y 373.273,Z 243.735,A -85,B 0,C 180,E1 -17285.842,E2 -17285.842} C_VEL
LIN {X 0,Y 376.455,Z 245.92,A -85,B 0,C 180,E1 -17291.025,E2 -17291.025} C_VEL
LIN {X 0,Y 376.938,Z 248.999,A -85,B 0,C 180,E1 -17292.097,E2 -17292.097} C_VEL
LIN {X 0,Y 377.372,Z 250.956,A -85,B 0,C 180,E1 -17292.824,E2 -17292.824} C_VEL
LIN {X 0,Y 378.09,Z 252.989,A -85,B 0,C 180,E1 -17293.613,E2 -17293.613} C_VEL
LIN {X 0,Y 381.942,Z 260.443,A -85,B 0,C 180,E1 -17295.643,E2 -17295.643} C_VEL
LIN {X 0,Y 386.64,Z 269.178,A -85,B 0,C 180,E1 -17297.924,E2 -17297.924} C_VEL
LIN {X 0,Y 393.585,Z 282.568,A -85,B 0,C 180,E1 -17301.146,E2 -17301.146} C_VEL
LIN {X 0,Y 401.935,Z 299.062,A -85,B 0,C 180,E1 -17304.769,E2 -17304.769} C_VEL
LIN {X 0,Y 410.782,Z 317.019,A -85,B 0,C 180,E1 -17308.337,E2 -17308.337} C_VEL
LIN {X 0,Y 417.869,Z 331.617,A -85,B 0,C 180,E1 -17310.941,E2 -17310.941} C_VEL
LIN {X 0,Y 436.305,Z 360.278,A -85,B 0,C 180,E1 -17314.059,E2 -17314.059} C_VEL
LIN {X 0,Y 442.82,Z 370.929,A -85,B 0,C 180,E1 -17315.098,E2 -17315.098} C_VEL
LIN {X 0,Y 425.049,Z 615.432,A -85,B 0,C 180,E1 -17320.148,E2 -17320.148} C_VEL
LIN {X 0,Y 419.838,Z 693.71,A -85,B 0,C 180,E1 -17321.829,E2 -17321.829} C_VEL
LIN {X 0,Y 417.204,Z 717.985,A -85,B 0,C 180,E1 -17322.566,E2 -17322.566} C_VEL
LIN {X 0,Y 413.793,Z 743.335,A -85,B 0,C 180,E1 -17323.581,E2 -17323.581} C_VEL
LIN {X 0,Y 410.214,Z 765.969,A -85,B 0,C 180,E1 -17324.722,E2 -17324.722} C_VEL
LIN {X 0,Y 406.115,Z 788.494,A -85,B 0,C 180,E1 -17326.126,E2 -17326.126} C_VEL
LIN {X 0,Y 401.696,Z 810.64,A -85,B 0,C 180,E1 -17327.773,E2 -17327.773} C_VEL
LIN {X 0,Y 397.243,Z 831.201,A -85,B 0,C 180,E1 -17329.598,E2 -17329.598} C_VEL
LIN {X 0,Y 392.5,Z 851.807,A -85,B 0,C 180,E1 -17331.754,E2 -17331.754} C_VEL
LIN {X 0,Y 388.001,Z 870.876,A -85,B 0,C 180,E1 -17334.085,E2 -17334.085} C_VEL
LIN {X 0,Y 383.726,Z 888.522,A -85,B 0,C 180,E1 -17336.646,E2 -17336.646} C_VEL
LIN {X 0,Y 379.566,Z 906.051,A -85,B 0,C 180,E1 -17339.617,E2 -17339.617} C_VEL
LIN {X 0,Y 376.502,Z 919.634,A -85,B 0,C 180,E1 -17342.306,E2 -17342.306} C_VEL
LIN {X 0,Y 373.64,Z 933.36,A -85,B 0,C 180,E1 -17345.494,E2 -17345.494} C_VEL
LIN {X 0,Y 371.584,Z 944.731,A -85,B 0,C 180,E1 -17348.599,E2 -17348.599} C_VEL
LIN {X 0,Y 370.123,Z 954.76,A -85,B 0,C 180,E1 -17351.9,E2 -17351.9} C_VEL
LIN {X 0,Y 369.274,Z 963.009,A -85,B 0,C 180,E1 -17355.163,E2 -17355.163} C_VEL
LIN {X 0,Y 368.9,Z 969.788,A -85,B 0,C 180,E1 -17358.588,E2 -17358.588} C_VEL
LIN {X 0,Y 368.885,Z 974.143,A -85,B 0,C 180,E1 -17361.426,E2 -17361.426} C_VEL
LIN {X 0,Y 369.026,Z 977.784,A -85,B 0,C 180,E1 -17364.714,E2 -17364.714} C_VEL
LIN {X 0,Y 369.163,Z 979.66,A -85,B 0,C 180,E1 -17367.827,E2 -17367.827} C_VEL
LIN {X 0,Y 369.166,Z 980.199,A -85,B 0,C 180,E1 -17370.621,E2 -17370.621} C_VEL
LIN {X 0,Y 369.057,Z 979.635,A -85,B 0,C 180,E1 -17373.417,E2 -17373.417} C_VEL
LIN {X 0,Y 368.807,Z 977.464,A -85,B 0,C 180,E1 -17376.851,E2 -17376.851} C_VEL
LIN {X 0,Y 368.697,Z 973.817,A -85,B 0,C 180,E1 -17380.153,E2 -17380.153} C_VEL
LIN {X 0,Y 368.887,Z 968.537,A -85,B 0,C 180,E1 -17383.64,E2 -17383.64} C_VEL
LIN {X 0,Y 369.681,Z 961.169,A -85,B 0,C 180,E1 -17387.309,E2 -17387.309} C_VEL
LIN {X 0,Y 371.108,Z 952.958,A -85,B 0,C 180,E1 -17390.669,E2 -17390.669} C_VEL
LIN {X 0,Y 373.613,Z 942.104,A -85,B 0,C 180,E1 -17394.34,E2 -17394.34} C_VEL
LIN {X 0,Y 377.059,Z 929.949,A -85,B 0,C 180,E1 -17397.822,E2 -17397.822} C_VEL
LIN {X 0,Y 381.621,Z 915.732,A -85,B 0,C 180,E1 -17401.251,E2 -17401.251} C_VEL
LIN {X 0,Y 387.402,Z 899.481,A -85,B 0,C 180,E1 -17404.599,E2 -17404.599} C_VEL
LIN {X 0,Y 393.749,Z 882.654,A -85,B 0,C 180,E1 -17407.55,E2 -17407.55} C_VEL
LIN {X 0,Y 401.166,Z 863.625,A -85,B 0,C 180,E1 -17410.394,E2 -17410.394} C_VEL
LIN {X 0,Y 409.288,Z 843.31,A -85,B 0,C 180,E1 -17412.969,E2 -17412.969} C_VEL
LIN {X 0,Y 417.921,Z 821.672,A -85,B 0,C 180,E1 -17415.283,E2 -17415.283} C_VEL
LIN {X 0,Y 427.008,Z 798.545,A -85,B 0,C 180,E1 -17417.33,E2 -17417.33} C_VEL
LIN {X 0,Y 436.125,Z 774.699,A -85,B 0,C 180,E1 -17419.064,E2 -17419.064} C_VEL
LIN {X 0,Y 445.112,Z 750.099,A -85,B 0,C 180,E1 -17420.501,E2 -17420.501} C_VEL
LIN {X 0,Y 453.088,Z 726.812,A -85,B 0,C 180,E1 -17421.576,E2 -17421.576} C_VEL
LIN {X 0,Y 458.046,Z 711.057,A -85,B 0,C 180,E1 -17422.163,E2 -17422.163} C_VEL
LIN {X 0,Y 449.744,Z 732.033,A -85,B 0,C 180,E1 -17423.11,E2 -17423.11} C_VEL
LIN {X 0,Y 440.64,Z 752.821,A -85,B 0,C 180,E1 -17424.325,E2 -17424.325} C_VEL
LIN {X 0,Y 431.017,Z 773.396,A -85,B 0,C 180,E1 -17425.847,E2 -17425.847} C_VEL
LIN {X 0,Y 421.296,Z 793.853,A -85,B 0,C 180,E1 -17427.723,E2 -17427.723} C_VEL
LIN {X 0,Y 412.313,Z 813.002,A -85,B 0,C 180,E1 -17429.868,E2 -17429.868} C_VEL
LIN {X 0,Y 404.141,Z 830.82,A -85,B 0,C 180,E1 -17432.281,E2 -17432.281} C_VEL
LIN {X 0,Y 397.131,Z 846.339,A -85,B 0,C 180,E1 -17434.817,E2 -17434.817} C_VEL
LIN {X 0,Y 391.155,Z 859.621,A -85,B 0,C 180,E1 -17437.453,E2 -17437.453} C_VEL
LIN {X 0,Y 386.349,Z 870.2,A -85,B 0,C 180,E1 -17440.024,E2 -17440.024} C_VEL
LIN {X 0,Y 382.158,Z 879.13,A -85,B 0,C 180,E1 -17442.746,E2 -17442.746} C_VEL
LIN {X 0,Y 378.757,Z 886.02,A -85,B 0,C 180,E1 -17445.476,E2 -17445.476} C_VEL
LIN {X 0,Y 375.938,Z 891.148,A -85,B 0,C 180,E1 -17448.338,E2 -17448.338} C_VEL
LIN {X 0,Y 373.877,Z 894.196,A -85,B 0,C 180,E1 -17451.077,E2 -17451.077} C_VEL
LIN {X 0,Y 372.344,Z 895.519,A -85,B 0,C 180,E1 -17453.834,E2 -17453.834} C_VEL
LIN {X 0,Y 371.268,Z 895.139,A -85,B 0,C 180,E1 -17456.603,E2 -17456.603} C_VEL
LIN {X 0,Y 370.597,Z 893.05,A -85,B 0,C 180,E1 -17459.382,E2 -17459.382} C_VEL
LIN {X 0,Y 370.227,Z 888.959,A -85,B 0,C 180,E1 -17462.322,E2 -17462.322} C_VEL
LIN {X 0,Y 370.195,Z 883.259,A -85,B 0,C 180,E1 -17465.114,E2 -17465.114} C_VEL
LIN {X 0,Y 370.477,Z 875.638,A -85,B 0,C 180,E1 -17467.912,E2 -17467.912} C_VEL
LIN {X 0,Y 371.115,Z 865.96,A -85,B 0,C 180,E1 -17470.714,E2 -17470.714} C_VEL
LIN {X 0,Y 372.157,Z 854.294,A -85,B 0,C 180,E1 -17473.443,E2 -17473.443} C_VEL
LIN {X 0,Y 373.557,Z 841.04,A -85,B 0,C 180,E1 -17476.004,E2 -17476.004} C_VEL
LIN {X 0,Y 375.292,Z 826.18,A -85,B 0,C 180,E1 -17478.404,E2 -17478.404} C_VEL
LIN {X 0,Y 377.313,Z 809.736,A -85,B 0,C 180,E1 -17480.638,E2 -17480.638} C_VEL
LIN {X 0,Y 379.573,Z 791.584,A -85,B 0,C 180,E1 -17482.701,E2 -17482.701} C_VEL
LIN {X 0,Y 381.887,Z 772.406,A -85,B 0,C 180,E1 -17484.519,E2 -17484.519} C_VEL
LIN {X 0,Y 384.23,Z 752.327,A -85,B 0,C 180,E1 -17486.091,E2 -17486.091} C_VEL
LIN {X 0,Y 386.651,Z 729.773,A -85,B 0,C 180,E1 -17487.522,E2 -17487.522} C_VEL
LIN {X 0,Y 388.821,Z 706.949,A -85,B 0,C 180,E1 -17488.66,E2 -17488.66} C_VEL
LIN {X 0,Y 390.726,Z 683.562,A -85,B 0,C 180,E1 -17489.527,E2 -17489.527} C_VEL
LIN {X 0,Y 402.308,Z 510.821,A -85,B 0,C 180,E1 -17494.109,E2 -17494.109} C_VEL
LIN {X 0,Y 398.01,Z 433.158,A -85,B 0,C 180,E1 -17497.018,E2 -17497.018} C_VEL
LIN {X 0,Y 399.122,Z 425.775,A -85,B 0,C 180,E1 -17497.682,E2 -17497.682} C_VEL
LIN {X 0,Y 400.794,Z 425.672,A -85,B 0,C 180,E1 -17498.04,E2 -17498.04} C_VEL
LIN {X 0,Y 404.192,Z 423.194,A -85,B 0,C 180,E1 -17498.565,E2 -17498.565} C_VEL
LIN {X 0,Y 408.518,Z 418.349,A -85,B 0,C 180,E1 -17499.069,E2 -17499.069} C_VEL
LIN {X 0,Y 412.157,Z 416.376,A -85,B 0,C 180,E1 -17499.646,E2 -17499.646} C_VEL
LIN {X 0,Y 416.658,Z 412.281,A -85,B 0,C 180,E1 -17500.207,E2 -17500.207} C_VEL
LIN {X 0,Y 418.233,Z 410.69,A -85,B 0,C 180,E1 -17500.383,E2 -17500.383} C_VEL
LIN {X 0,Y 423.151,Z 407.544,A -85,B 0,C 180,E1 -17501.064,E2 -17501.064} C_VEL
LIN {X 0,Y 427.767,Z 403.435,A -85,B 0,C 180,E1 -17501.594,E2 -17501.594} C_VEL
LIN {X 0,Y 433.627,Z 399.518,A -85,B 0,C 180,E1 -17502.324,E2 -17502.324} C_VEL
LIN {X 0,Y 436.753,Z 396.908,A -85,B 0,C 180,E1 -17502.661,E2 -17502.661} C_VEL
LIN {X 0,Y 439.482,Z 395.295,A -85,B 0,C 180,E1 -17503,E2 -17503} C_VEL
LIN {X 0,Y 436.048,Z 411.878,A -85,B 0,C 180,E1 -17503.573,E2 -17503.573} C_VEL
LIN {X 0,Y 431.592,Z 491.845,A -85,B 0,C 180,E1 -17504.956,E2 -17504.956} C_VEL
LIN {X 0,Y 426.935,Z 551.477,A -85,B 0,C 180,E1 -17506.206,E2 -17506.206} C_VEL
LIN {X 0,Y 421.004,Z 612.454,A -85,B 0,C 180,E1 -17507.717,E2 -17507.717} C_VEL
LIN {X 0,Y 416.613,Z 656.627,A -85,B 0,C 180,E1 -17509.024,E2 -17509.024} C_VEL
LIN {X 0,Y 414.143,Z 684.167,A -85,B 0,C 180,E1 -17510.031,E2 -17510.031} C_VEL
LIN {X 0,Y 411.671,Z 704.67,A -85,B 0,C 180,E1 -17511.018,E2 -17511.018} C_VEL
LIN {X 0,Y 408.494,Z 725.351,A -85,B 0,C 180,E1 -17512.27,E2 -17512.27} C_VEL
LIN {X 0,Y 404.886,Z 745.039,A -85,B 0,C 180,E1 -17513.739,E2 -17513.739} C_VEL
LIN {X 0,Y 400.919,Z 763.783,A -85,B 0,C 180,E1 -17515.432,E2 -17515.432} C_VEL
LIN {X 0,Y 396.544,Z 782.178,A -85,B 0,C 180,E1 -17517.429,E2 -17517.429} C_VEL
LIN {X 0,Y 392.084,Z 799.399,A -85,B 0,C 180,E1 -17519.673,E2 -17519.673} C_VEL
LIN {X 0,Y 387.682,Z 815.388,A -85,B 0,C 180,E1 -17522.171,E2 -17522.171} C_VEL
LIN {X 0,Y 383.596,Z 829.715,A -85,B 0,C 180,E1 -17524.857,E2 -17524.857} C_VEL
LIN {X 0,Y 379.924,Z 842.44,A -85,B 0,C 180,E1 -17527.729,E2 -17527.729} C_VEL
LIN {X 0,Y 376.762,Z 853.567,A -85,B 0,C 180,E1 -17530.787,E2 -17530.787} C_VEL
LIN {X 0,Y 374.193,Z 863.077,A -85,B 0,C 180,E1 -17534.024,E2 -17534.024} C_VEL
LIN {X 0,Y 372.324,Z 870.574,A -85,B 0,C 180,E1 -17537.278,E2 -17537.278} C_VEL
LIN {X 0,Y 371.08,Z 876.131,A -85,B 0,C 180,E1 -17540.473,E2 -17540.473} C_VEL
LIN {X 0,Y 370.852,Z 877.297,A -85,B 0,C 180,E1 -17541.273,E2 -17541.273} C_VEL
LIN {X 0,Y 369.576,Z 878.907,A -85,B 0,C 180,E1 -17542.434,E2 -17542.434} C_VEL
LIN {X 0,Y 362.889,Z 882.676,A -85,B 0,C 180,E1 -17545.54,E2 -17545.54} C_VEL
LIN {X 0,Y 362.034,Z 883.325,A -85,B 0,C 180,E1 -17546.583,E2 -17546.583} C_VEL
LIN {X 0,Y 361.899,Z 884.203,A -85,B 0,C 180,E1 -17549.842,E2 -17549.842} C_VEL
LIN {X 0,Y 361.99,Z 883.531,A -85,B 0,C 180,E1 -17553.008,E2 -17553.008} C_VEL
LIN {X 0,Y 362.391,Z 881.282,A -85,B 0,C 180,E1 -17556.336,E2 -17556.336} C_VEL
LIN {X 0,Y 363.134,Z 877.643,A -85,B 0,C 180,E1 -17559.509,E2 -17559.509} C_VEL
LIN {X 0,Y 364.434,Z 872.141,A -85,B 0,C 180,E1 -17562.84,E2 -17562.84} C_VEL
LIN {X 0,Y 366.359,Z 864.769,A -85,B 0,C 180,E1 -17566.164,E2 -17566.164} C_VEL
LIN {X 0,Y 369.008,Z 855.422,A -85,B 0,C 180,E1 -17569.468,E2 -17569.468} C_VEL
LIN {X 0,Y 372.088,Z 845.046,A -85,B 0,C 180,E1 -17572.432,E2 -17572.432} C_VEL
LIN {X 0,Y 375.623,Z 833.33,A -85,B 0,C 180,E1 -17575.208,E2 -17575.208} C_VEL
LIN {X 0,Y 379.769,Z 819.481,A -85,B 0,C 180,E1 -17577.947,E2 -17577.947} C_VEL
LIN {X 0,Y 384.109,Z 804.526,A -85,B 0,C 180,E1 -17580.418,E2 -17580.418} C_VEL
LIN {X 0,Y 388.694,Z 787.801,A -85,B 0,C 180,E1 -17582.734,E2 -17582.734} C_VEL
LIN {X 0,Y 393.15,Z 770.226,A -85,B 0,C 180,E1 -17584.766,E2 -17584.766} C_VEL
LIN {X 0,Y 397.486,Z 751.2,A -85,B 0,C 180,E1 -17586.597,E2 -17586.597} C_VEL
LIN {X 0,Y 401.362,Z 731.573,A -85,B 0,C 180,E1 -17588.158,E2 -17588.158} C_VEL
LIN {X 0,Y 404.643,Z 712.102,A -85,B 0,C 180,E1 -17589.424,E2 -17589.424} C_VEL
LIN {X 0,Y 407.411,Z 691.583,A -85,B 0,C 180,E1 -17590.501,E2 -17590.501} C_VEL
LIN {X 0,Y 409.614,Z 669.832,A -85,B 0,C 180,E1 -17591.381,E2 -17591.381} C_VEL
LIN {X 0,Y 413.811,Z 626.601,A -85,B 0,C 180,E1 -17592.758,E2 -17592.758} C_VEL
LIN {X 0,Y 419.839,Z 568.778,A -85,B 0,C 180,E1 -17594.269,E2 -17594.269} C_VEL
